LIN {X 0,Y 362.968,Z 415.154,A -85,B 0,C 180,E1 -13446.297,E2 -13446.297} C_VEL
LIN {X 0,Y 357.629,Z 396.824,A -85,B 0,C 180,E1 -13449.531,E2 -13449.531} C_VEL
LIN {X 0,Y 354.805,Z 387.089,A -85,B 0,C 180,E1 -13451.373,E2 -13451.373} C_VEL
LIN {X 0,Y 354.749,Z 386.923,A -85,B 0,C 180,E1 -13454.504,E2 -13454.504} C_VEL
LIN {X 0,Y 354.769,Z 386.876,A -85,B 0,C 180,E1 -13457.659,E2 -13457.659} C_VEL
LIN {X 0,Y 354.773,Z 386.917,A -85,B 0,C 180,E1 -13460.661,E2 -13460.661} C_VEL
LIN {X 0,Y 354.805,Z 386.863,A -85,B 0,C 180,E1 -13464.301,E2 -13464.301} C_VEL
LIN {X 0,Y 354.773,Z 386.912,A -85,B 0,C 180,E1 -13467.665,E2 -13467.665} C_VEL
LIN {X 0,Y 354.785,Z 386.907,A -85,B 0,C 180,E1 -13471.613,E2 -13471.613} C_VEL
LIN {X 0,Y 354.79,Z 386.899,A -85,B 0,C 180,E1 -13475.419,E2 -13475.419} C_VEL
LIN {X 0,Y 354.809,Z 386.903,A -85,B 0,C 180,E1 -13479.112,E2 -13479.112} C_VEL
LIN {X 0,Y 354.836,Z 386.911,A -85,B 0,C 180,E1 -13482.717,E2 -13482.717} C_VEL
LIN {X 0,Y 354.924,Z 386.887,A -85,B 0,C 180,E1 -13486.254,E2 -13486.254} C_VEL
LIN {X 0,Y 354.937,Z 386.882,A -85,B 0,C 180,E1 -13489.735,E2 -13489.735} C_VEL
LIN {X 0,Y 355.066,Z 386.879,A -85,B 0,C 180,E1 -13493.18,E2 -13493.18} C_VEL
LIN {X 0,Y 355.214,Z 386.859,A -85,B 0,C 180,E1 -13497.732,E2 -13497.732} C_VEL
LIN {X 0,Y 355.212,Z 386.849,A -85,B 0,C 180,E1 -13502.268,E2 -13502.268} C_VEL
LIN {X 0,Y 355.089,Z 386.861,A -85,B 0,C 180,E1 -13506.82,E2 -13506.82} C_VEL
LIN {X 0,Y 354.939,Z 386.89,A -85,B 0,C 180,E1 -13510.265,E2 -13510.265} C_VEL
LIN {X 0,Y 354.928,Z 386.895,A -85,B 0,C 180,E1 -13514.019,E2 -13514.019} C_VEL
LIN {X 0,Y 354.876,Z 386.898,A -85,B 0,C 180,E1 -13518.093,E2 -13518.093} C_VEL
LIN {X 0,Y 354.793,Z 386.906,A -85,B 0,C 180,E1 -13522.109,E2 -13522.109} C_VEL
LIN {X 0,Y 354.787,Z 386.904,A -85,B 0,C 180,E1 -13525.836,E2 -13525.836} C_VEL
LIN {X 0,Y 354.78,Z 386.909,A -85,B 0,C 180,E1 -13529.686,E2 -13529.686} C_VEL
LIN {X 0,Y 354.795,Z 386.915,A -85,B 0,C 180,E1 -13533.703,E2 -13533.703} C_VEL
LIN {X 0,Y 354.78,Z 386.888,A -85,B 0,C 180,E1 -13536.462,E2 -13536.462} C_VEL
LIN {X 0,Y 354.757,Z 386.91,A -85,B 0,C 180,E1 -13539.414,E2 -13539.414} C_VEL
LIN {X 0,Y 354.769,Z 386.891,A -85,B 0,C 180,E1 -13542.867,E2 -13542.867} C_VEL
LIN {X 0,Y 354.797,Z 387.142,A -85,B 0,C 180,E1 -13544.912,E2 -13544.912} C_VEL
LIN {X 0,Y 357.139,Z 393.195,A -85,B 0,C 180,E1 -13546.219,E2 -13546.219} C_VEL
LIN {X 0,Y 362.106,Z 406.376,A -85,B 0,C 180,E1 -13548.824,E2 -13548.824} C_VEL
LIN {X 0,Y 366.575,Z 420.211,A -85,B 0,C 180,E1 -13551.376,E2 -13551.376} C_VEL
LIN {X 0,Y 370.495,Z 434.136,A -85,B 0,C 180,E1 -13553.779,E2 -13553.779} C_VEL
LIN {X 0,Y 371.189,Z 437.502,A -85,B 0,C 180,E1 -13554.317,E2 -13554.317} C_VEL
LIN {X 0,Y 369.064,Z 461.57,A -85,B 0,C 180,E1 -13557.353,E2 -13557.353} C_VEL
LIN {X 0,Y 368.412,Z 471.572,A -85,B 0,C 180,E1 -13558.53,E2 -13558.53} C_VEL
LIN {X 0,Y 373.171,Z 501.555,A -85,B 0,C 180,E1 -13559.641,E2 -13559.641} C_VEL
LIN {X 0,Y 374.104,Z 509.019,A -85,B 0,C 180,E1 -13559.887,E2 -13559.887} C_VEL
LIN {X 0,Y 370.581,Z 640.588,A -85,B 0,C 180,E1 -13562.469,E2 -13562.469} C_VEL
LIN {X 0,Y 369.736,Z 655.386,A -85,B 0,C 180,E1 -13562.945,E2 -13562.945} C_VEL
LIN {X 0,Y 368.618,Z 669.241,A -85,B 0,C 180,E1 -13563.582,E2 -13563.582} C_VEL
LIN {X 0,Y 367.111,Z 684.092,A -85,B 0,C 180,E1 -13564.497,E2 -13564.497} C_VEL
LIN {X 0,Y 365.467,Z 697.803,A -85,B 0,C 180,E1 -13565.581,E2 -13565.581} C_VEL
LIN {X 0,Y 363.7,Z 710.491,A -85,B 0,C 180,E1 -13566.816,E2 -13566.816} C_VEL
LIN {X 0,Y 361.771,Z 723.288,A -85,B 0,C 180,E1 -13568.342,E2 -13568.342} C_VEL
LIN {X 0,Y 359.982,Z 734.883,A -85,B 0,C 180,E1 -13570.024,E2 -13570.024} C_VEL
LIN {X 0,Y 358.316,Z 744.651,A -85,B 0,C 180,E1 -13571.712,E2 -13571.712} C_VEL
LIN {X 0,Y 356.802,Z 754.205,A -85,B 0,C 180,E1 -13573.701,E2 -13573.701} C_VEL
LIN {X 0,Y 355.593,Z 762.353,A -85,B 0,C 180,E1 -13575.754,E2 -13575.754} C_VEL
LIN {X 0,Y 354.609,Z 769.585,A -85,B 0,C 180,E1 -13577.991,E2 -13577.991} C_VEL
LIN {X 0,Y 353.878,Z 775.478,A -85,B 0,C 180,E1 -13580.283,E2 -13580.283} C_VEL
LIN {X 0,Y 353.528,Z 778.954,A -85,B 0,C 180,E1 -13582.003,E2 -13582.003} C_VEL
LIN {X 0,Y 353.26,Z 782.496,A -85,B 0,C 180,E1 -13584.293,E2 -13584.293} C_VEL
LIN {X 0,Y 353.184,Z 784.838,A -85,B 0,C 180,E1 -13586.579,E2 -13586.579} C_VEL
LIN {X 0,Y 353.144,Z 786.03,A -85,B 0,C 180,E1 -13588.861,E2 -13588.861} C_VEL
LIN {X 0,Y 353.145,Z 786.044,A -85,B 0,C 180,E1 -13591.142,E2 -13591.142} C_VEL
LIN {X 0,Y 353.186,Z 784.909,A -85,B 0,C 180,E1 -13593.424,E2 -13593.424} C_VEL
LIN {X 0,Y 353.315,Z 782.299,A -85,B 0,C 180,E1 -13595.967,E2 -13595.967} C_VEL
LIN {X 0,Y 353.646,Z 778.076,A -85,B 0,C 180,E1 -13598.573,E2 -13598.573} C_VEL
LIN {X 0,Y 354.128,Z 772.946,A -85,B 0,C 180,E1 -13600.869,E2 -13600.869} C_VEL
LIN {X 0,Y 355.058,Z 766.383,A -85,B 0,C 180,E1 -13603.159,E2 -13603.159} C_VEL
LIN {X 0,Y 355.51,Z 763.086,A -85,B 0,C 180,E1 -13604.138,E2 -13604.138} C_VEL
LIN {X 0,Y 355.295,Z 760.19,A -85,B 0,C 180,E1 -13604.968,E2 -13604.968} C_VEL
LIN {X 0,Y 353.242,Z 755.303,A -85,B 0,C 180,E1 -13606.325,E2 -13606.325} C_VEL
LIN {X 0,Y 351.29,Z 749.969,A -85,B 0,C 180,E1 -13607.649,E2 -13607.649} C_VEL
LIN {X 0,Y 351.23,Z 746.373,A -85,B 0,C 180,E1 -13608.414,E2 -13608.414} C_VEL
LIN {X 0,Y 353.087,Z 735.857,A -85,B 0,C 180,E1 -13610.314,E2 -13610.314} C_VEL
LIN {X 0,Y 355.017,Z 723.948,A -85,B 0,C 180,E1 -13612.096,E2 -13612.096} C_VEL
LIN {X 0,Y 357.067,Z 711.288,A -85,B 0,C 180,E1 -13613.644,E2 -13613.644} C_VEL
LIN {X 0,Y 358.867,Z 698.787,A -85,B 0,C 180,E1 -13614.903,E2 -13614.903} C_VEL
LIN {X 0,Y 360.715,Z 684.652,A -85,B 0,C 180,E1 -13616.046,E2 -13616.046} C_VEL
LIN {X 0,Y 362.175,Z 670.066,A -85,B 0,C 180,E1 -13616.975,E2 -13616.975} C_VEL
LIN {X 0,Y 363.457,Z 655.655,A -85,B 0,C 180,E1 -13617.652,E2 -13617.652} C_VEL
LIN {X 0,Y 364.353,Z 639.939,A -85,B 0,C 180,E1 -13618.164,E2 -13618.164} C_VEL
LIN {X 0,Y 367.302,Z 535.361,A -85,B 0,C 180,E1 -13620.246,E2 -13620.246} C_VEL
LIN {X 0,Y 367.924,Z 508.361,A -85,B 0,C 180,E1 -13620.791,E2 -13620.791} C_VEL
LIN {X 0,Y 362.697,Z 474.811,A -85,B 0,C 180,E1 -13622.047,E2 -13622.047} C_VEL
LIN {X 0,Y 362.119,Z 471.033,A -85,B 0,C 180,E1 -13622.221,E2 -13622.221} C_VEL
LIN {X 0,Y 364.049,Z 448.22,A -85,B 0,C 180,E1 -13625.054,E2 -13625.054} C_VEL
LIN {X 0,Y 364.792,Z 439.692,A -85,B 0,C 180,E1 -13626.166,E2 -13626.166} C_VEL
LIN {X 0,Y 361.536,Z 427.166,A -85,B 0,C 180,E1 -13628.32,E2 -13628.32} C_VEL
LIN {X 0,Y 357.787,Z 414.84,A -85,B 0,C 180,E1 -13630.571,E2 -13630.571} C_VEL
LIN {X 0,Y 352.853,Z 400.954,A -85,B 0,C 180,E1 -13633.326,E2 -13633.326} C_VEL
LIN {X 0,Y 347.745,Z 388.016,A -85,B 0,C 180,E1 -13636.095,E2 -13636.095} C_VEL
LIN {X 0,Y 347.712,Z 387.785,A -85,B 0,C 180,E1 -13638.406,E2 -13638.406} C_VEL
LIN {X 0,Y 347.766,Z 387.788,A -85,B 0,C 180,E1 -13642.015,E2 -13642.015} C_VEL
LIN {X 0,Y 347.748,Z 387.758,A -85,B 0,C 180,E1 -13645.536,E2 -13645.536} C_VEL
LIN {X 0,Y 347.735,Z 387.795,A -85,B 0,C 180,E1 -13648.299,E2 -13648.299} C_VEL
LIN {X 0,Y 347.746,Z 387.792,A -85,B 0,C 180,E1 -13650.985,E2 -13650.985} C_VEL
LIN {X 0,Y 347.793,Z 387.981,A -85,B 0,C 180,E1 -13652.376,E2 -13652.376} C_VEL
LIN {X 0,Y 348.722,Z 391.932,A -85,B 0,C 180,E1 -13653.247,E2 -13653.247} C_VEL
LIN {X 0,Y 359.484,Z 420.146,A -85,B 0,C 180,E1 -13654.74,E2 -13654.74} C_VEL
LIN {X 0,Y 355.715,Z 535.123,A -85,B 0,C 180,E1 -13657.837,E2 -13657.837} C_VEL
LIN {X 0,Y 355.227,Z 550.727,A -85,B 0,C 180,E1 -13658.488,E2 -13658.488} C_VEL
LIN {X 0,Y 354.603,Z 565.332,A -85,B 0,C 180,E1 -13659.327,E2 -13659.327} C_VEL
LIN {X 0,Y 353.691,Z 579.963,A -85,B 0,C 180,E1 -13660.408,E2 -13660.408} C_VEL
LIN {X 0,Y 352.843,Z 593.82,A -85,B 0,C 180,E1 -13661.717,E2 -13661.717} C_VEL
LIN {X 0,Y 351.84,Z 606.827,A -85,B 0,C 180,E1 -13663.223,E2 -13663.223} C_VEL
LIN {X 0,Y 351.135,Z 616.893,A -85,B 0,C 180,E1 -13664.628,E2 -13664.628} C_VEL
LIN {X 0,Y 350.183,Z 627.379,A -85,B 0,C 180,E1 -13666.36,E2 -13666.36} C_VEL
LIN {X 0,Y 349.57,Z 636.146,A -85,B 0,C 180,E1 -13668.108,E2 -13668.108} C_VEL
LIN {X 0,Y 348.967,Z 644.601,A -85,B 0,C 180,E1 -13670.143,E2 -13670.143} C_VEL
LIN {X 0,Y 348.594,Z 650.5,A -85,B 0,C 180,E1 -13671.887,E2 -13671.887} C_VEL
LIN {X 0,Y 348.334,Z 655.341,A -85,B 0,C 180,E1 -13673.629,E2 -13673.629} C_VEL
LIN {X 0,Y 347.977,Z 660.381,A -85,B 0,C 180,E1 -13675.946,E2 -13675.946} C_VEL
LIN {X 0,Y 347.967,Z 663.099,A -85,B 0,C 180,E1 -13677.685,E2 -13677.685} C_VEL
LIN {X 0,Y 348.047,Z 665.484,A -85,B 0,C 180,E1 -13680,E2 -13680} C_VEL
LIN {X 0,Y 348.502,Z 666.421,A -85,B 0,C 180,E1 -13682.311,E2 -13682.311} C_VEL
LIN {X 0,Y 349.06,Z 665.935,A -85,B 0,C 180,E1 -13684.619,E2 -13684.619} C_VEL
LIN {X 0,Y 349.703,Z 664.039,A -85,B 0,C 180,E1 -13686.926,E2 -13686.926} C_VEL
LIN {X 0,Y 350.82,Z 660.596,A -85,B 0,C 180,E1 -13689.222,E2 -13689.222} C_VEL
LIN {X 0,Y 351.834,Z 657.006,A -85,B 0,C 180,E1 -13690.939,E2 -13690.939} C_VEL
LIN {X 0,Y 353.413,Z 650.686,A -85,B 0,C 180,E1 -13693.22,E2 -13693.22} C_VEL
LIN {X 0,Y 354.959,Z 643.625,A -85,B 0,C 180,E1 -13695.209,E2 -13695.209} C_VEL
LIN {X 0,Y 356.859,Z 634.78,A -85,B 0,C 180,E1 -13697.182,E2 -13697.182} C_VEL
LIN {X 0,Y 358.664,Z 625.61,A -85,B 0,C 180,E1 -13698.864,E2 -13698.864} C_VEL
LIN {X 0,Y 360.446,Z 615.653,A -85,B 0,C 180,E1 -13700.368,E2 -13700.368} C_VEL
LIN {X 0,Y 362.343,Z 603.197,A -85,B 0,C 180,E1 -13701.924,E2 -13701.924} C_VEL
LIN {X 0,Y 364.021,Z 591.036,A -85,B 0,C 180,E1 -13703.164,E2 -13703.164} C_VEL
LIN {X 0,Y 365.637,Z 577.686,A -85,B 0,C 180,E1 -13704.258,E2 -13704.258} C_VEL
LIN {X 0,Y 366.991,Z 564.198,A -85,B 0,C 180,E1 -13705.15,E2 -13705.15} C_VEL
LIN {X 0,Y 368.094,Z 548.734,A -85,B 0,C 180,E1 -13705.927,E2 -13705.927} C_VEL
LIN {X 0,Y 369.757,Z 525.884,A -85,B 0,C 180,E1 -13706.796,E2 -13706.796} C_VEL
LIN {X 0,Y 377.897,Z 451.52,A -85,B 0,C 180,E1 -13709.427,E2 -13709.427} C_VEL
LIN {X 0,Y 378.713,Z 443.174,A -85,B 0,C 180,E1 -13709.753,E2 -13709.753} C_VEL
LIN {X 0,Y 374.725,Z 436.391,A -85,B 0,C 180,E1 -13711.04,E2 -13711.04} C_VEL
LIN {X 0,Y 370.277,Z 430.062,A -85,B 0,C 180,E1 -13712.635,E2 -13712.635} C_VEL
LIN {X 0,Y 366.994,Z 426.007,A -85,B 0,C 180,E1 -13713.98,E2 -13713.98} C_VEL
LIN {X 0,Y 364.266,Z 422.895,A -85,B 0,C 180,E1 -13715.295,E2 -13715.295} C_VEL
LIN {X 0,Y 361.379,Z 419.769,A -85,B 0,C 180,E1 -13717.12,E2 -13717.12} C_VEL
LIN {X 0,Y 361.362,Z 419.182,A -85,B 0,C 180,E1 -13718.925,E2 -13718.925} C_VEL
LIN {X 0,Y 361.655,Z 419.554,A -85,B 0,C 180,E1 -13721.355,E2 -13721.355} C_VEL
LIN {X 0,Y 362.637,Z 421.568,A -85,B 0,C 180,E1 -13724.242,E2 -13724.242} C_VEL
LIN {X 0,Y 363.768,Z 424.413,A -85,B 0,C 180,E1 -13726.426,E2 -13726.426} C_VEL
LIN {X 0,Y 365.158,Z 428.525,A -85,B 0,C 180,E1 -13728.643,E2 -13728.643} C_VEL
LIN {X 0,Y 366.624,Z 433.697,A -85,B 0,C 180,E1 -13730.757,E2 -13730.757} C_VEL
LIN {X 0,Y 368.039,Z 439.973,A -85,B 0,C 180,E1 -13732.763,E2 -13732.763} C_VEL
LIN {X 0,Y 370.061,Z 445.463,A -85,B 0,C 180,E1 -13733.732,E2 -13733.732} C_VEL
LIN {X 0,Y 371.308,Z 455.894,A -85,B 0,C 180,E1 -13734.7,E2 -13734.7} C_VEL
LIN {X 0,Y 372.834,Z 472.254,A -85,B 0,C 180,E1 -13735.965,E2 -13735.965} C_VEL
LIN {X 0,Y 373.775,Z 487.634,A -85,B 0,C 180,E1 -13736.955,E2 -13736.955} C_VEL
LIN {X 0,Y 374.116,Z 504.327,A -85,B 0,C 180,E1 -13737.835,E2 -13737.835} C_VEL
LIN {X 0,Y 373.957,Z 509.719,A -85,B 0,C 180,E1 -13738.061,E2 -13738.061} C_VEL
LIN {X 0,Y 368.616,Z 574.67,A -85,B 0,C 180,E1 -13740.085,E2 -13740.085} C_VEL
LIN {X 0,Y 365.731,Z 612.624,A -85,B 0,C 180,E1 -13741.247,E2 -13741.247} C_VEL
LIN {X 0,Y 364.27,Z 626.12,A -85,B 0,C 180,E1 -13741.79,E2 -13741.79} C_VEL
LIN {X 0,Y 363.515,Z 645.43,A -85,B 0,C 180,E1 -13742.235,E2 -13742.235} C_VEL
LIN {X 0,Y 362.466,Z 660.753,A -85,B 0,C 180,E1 -13742.814,E2 -13742.814} C_VEL
LIN {X 0,Y 361.182,Z 674.979,A -85,B 0,C 180,E1 -13743.57,E2 -13743.57} C_VEL
LIN {X 0,Y 359.668,Z 688.894,A -85,B 0,C 180,E1 -13744.538,E2 -13744.538} C_VEL
LIN {X 0,Y 357.77,Z 703.113,A -85,B 0,C 180,E1 -13745.789,E2 -13745.789} C_VEL
LIN {X 0,Y 355.877,Z 715.961,A -85,B 0,C 180,E1 -13747.196,E2 -13747.196} C_VEL
LIN {X 0,Y 353.992,Z 727.703,A -85,B 0,C 180,E1 -13748.755,E2 -13748.755} C_VEL
LIN {X 0,Y 352.295,Z 738.439,A -85,B 0,C 180,E1 -13750.478,E2 -13750.478} C_VEL
LIN {X 0,Y 350.726,Z 747.527,A -85,B 0,C 180,E1 -13752.205,E2 -13752.205} C_VEL
LIN {X 0,Y 349.286,Z 756.423,A -85,B 0,C 180,E1 -13754.237,E2 -13754.237} C_VEL
LIN {X 0,Y 348.026,Z 764.73,A -85,B 0,C 180,E1 -13756.57,E2 -13756.57} C_VEL
LIN {X 0,Y 347.132,Z 771.379,A -85,B 0,C 180,E1 -13758.909,E2 -13758.909} C_VEL
LIN {X 0,Y 346.628,Z 776.575,A -85,B 0,C 180,E1 -13761.252,E2 -13761.252} C_VEL
LIN {X 0,Y 346.325,Z 780.853,A -85,B 0,C 180,E1 -13763.912,E2 -13763.912} C_VEL
LIN {X 0,Y 346.187,Z 783.505,A -85,B 0,C 180,E1 -13766.507,E2 -13766.507} C_VEL
LIN {X 0,Y 346.129,Z 784.673,A -85,B 0,C 180,E1 -13768.835,E2 -13768.835} C_VEL
LIN {X 0,Y 346.132,Z 784.671,A -85,B 0,C 180,E1 -13771.162,E2 -13771.162} C_VEL
LIN {X 0,Y 346.189,Z 783.496,A -85,B 0,C 180,E1 -13773.49,E2 -13773.49} C_VEL
LIN {X 0,Y 346.285,Z 780.913,A -85,B 0,C 180,E1 -13776.026,E2 -13776.026} C_VEL
LIN {X 0,Y 346.621,Z 776.563,A -85,B 0,C 180,E1 -13778.745,E2 -13778.745} C_VEL
LIN {X 0,Y 347.125,Z 771.36,A -85,B 0,C 180,E1 -13781.087,E2 -13781.087} C_VEL
LIN {X 0,Y 348.009,Z 764.698,A -85,B 0,C 180,E1 -13783.427,E2 -13783.427} C_VEL
LIN {X 0,Y 349.267,Z 756.386,A -85,B 0,C 180,E1 -13785.76,E2 -13785.76} C_VEL
LIN {X 0,Y 350.692,Z 747.486,A -85,B 0,C 180,E1 -13787.793,E2 -13787.793} C_VEL
LIN {X 0,Y 352.266,Z 738.387,A -85,B 0,C 180,E1 -13789.52,E2 -13789.52} C_VEL
LIN {X 0,Y 353.967,Z 727.642,A -85,B 0,C 180,E1 -13791.243,E2 -13791.243} C_VEL
LIN {X 0,Y 355.824,Z 715.892,A -85,B 0,C 180,E1 -13792.804,E2 -13792.804} C_VEL
LIN {X 0,Y 357.747,Z 703.017,A -85,B 0,C 180,E1 -13794.208,E2 -13794.208} C_VEL
LIN {X 0,Y 359.399,Z 690.514,A -85,B 0,C 180,E1 -13795.323,E2 -13795.323} C_VEL
LIN {X 0,Y 361.03,Z 676.025,A -85,B 0,C 180,E1 -13796.355,E2 -13796.355} C_VEL
LIN {X 0,Y 362.375,Z 661.307,A -85,B 0,C 180,E1 -13797.151,E2 -13797.151} C_VEL
LIN {X 0,Y 363.412,Z 646.234,A -85,B 0,C 180,E1 -13797.73,E2 -13797.73} C_VEL
LIN {X 0,Y 364.103,Z 629.144,A -85,B 0,C 180,E1 -13798.142,E2 -13798.142} C_VEL
LIN {X 0,Y 367.019,Z 518.003,A -85,B 0,C 180,E1 -13800.331,E2 -13800.331} C_VEL
LIN {X 0,Y 367.175,Z 504.545,A -85,B 0,C 180,E1 -13800.615,E2 -13800.615} C_VEL
LIN {X 0,Y 363.359,Z 473.493,A -85,B 0,C 180,E1 -13801.676,E2 -13801.676} C_VEL
LIN {X 0,Y 362.286,Z 465.651,A -85,B 0,C 180,E1 -13801.993,E2 -13801.993} C_VEL
LIN {X 0,Y 360.716,Z 438.296,A -85,B 0,C 180,E1 -13803.739,E2 -13803.739} C_VEL
LIN {X 0,Y 359.932,Z 430.462,A -85,B 0,C 180,E1 -13804.261,E2 -13804.261} C_VEL
LIN {X 0,Y 355.292,Z 413.79,A -85,B 0,C 180,E1 -13807.067,E2 -13807.067} C_VEL
LIN {X 0,Y 350.111,Z 396.023,A -85,B 0,C 180,E1 -13810.289,E2 -13810.289} C_VEL
LIN {X 0,Y 347.758,Z 387.949,A -85,B 0,C 180,E1 -13811.875,E2 -13811.875} C_VEL
LIN {X 0,Y 347.691,Z 387.801,A -85,B 0,C 180,E1 -13815.026,E2 -13815.026} C_VEL
LIN {X 0,Y 347.725,Z 387.754,A -85,B 0,C 180,E1 -13818.398,E2 -13818.398} C_VEL
LIN {X 0,Y 347.749,Z 387.784,A -85,B 0,C 180,E1 -13822.013,E2 -13822.013} C_VEL
LIN {X 0,Y 347.729,Z 387.746,A -85,B 0,C 180,E1 -13825.535,E2 -13825.535} C_VEL
LIN {X 0,Y 347.732,Z 387.794,A -85,B 0,C 180,E1 -13828.299,E2 -13828.299} C_VEL
LIN {X 0,Y 347.731,Z 387.781,A -85,B 0,C 180,E1 -13830.983,E2 -13830.983} C_VEL
LIN {X 0,Y 347.729,Z 387.794,A -85,B 0,C 180,E1 -13833.599,E2 -13833.599} C_VEL
LIN {X 0,Y 347.734,Z 387.782,A -85,B 0,C 180,E1 -13836.158,E2 -13836.158} C_VEL
LIN {X 0,Y 347.761,Z 387.774,A -85,B 0,C 180,E1 -13839.906,E2 -13839.906} C_VEL
LIN {X 0,Y 347.782,Z 387.786,A -85,B 0,C 180,E1 -13843.566,E2 -13843.566} C_VEL
LIN {X 0,Y 347.871,Z 387.777,A -85,B 0,C 180,E1 -13847.16,E2 -13847.16} C_VEL
LIN {X 0,Y 347.919,Z 387.753,A -85,B 0,C 180,E1 -13850.7,E2 -13850.7} C_VEL
LIN {X 0,Y 348.019,Z 387.752,A -85,B 0,C 180,E1 -13854.205,E2 -13854.205} C_VEL
LIN {X 0,Y 348.176,Z 387.735,A -85,B 0,C 180,E1 -13857.686,E2 -13857.686} C_VEL
LIN {X 0,Y 348.127,Z 387.725,A -85,B 0,C 180,E1 -13861.157,E2 -13861.157} C_VEL
LIN {X 0,Y 348.174,Z 387.726,A -85,B 0,C 180,E1 -13862.314,E2 -13862.314} C_VEL
LIN {X 0,Y 348.057,Z 387.736,A -85,B 0,C 180,E1 -13866.959,E2 -13866.959} C_VEL
LIN {X 0,Y 347.879,Z 387.765,A -85,B 0,C 180,E1 -13870.476,E2 -13870.476} C_VEL
LIN {X 0,Y 347.884,Z 387.773,A -85,B 0,C 180,E1 -13874.151,E2 -13874.151} C_VEL
LIN {X 0,Y 347.815,Z 387.779,A -85,B 0,C 180,E1 -13878.26,E2 -13878.26} C_VEL
LIN {X 0,Y 347.75,Z 387.778,A -85,B 0,C 180,E1 -13881.625,E2 -13881.625} C_VEL
LIN {X 0,Y 347.724,Z 387.783,A -85,B 0,C 180,E1 -13885.115,E2 -13885.115} C_VEL
LIN {X 0,Y 347.711,Z 387.798,A -85,B 0,C 180,E1 -13887.703,E2 -13887.703} C_VEL
LIN {X 0,Y 347.716,Z 387.794,A -85,B 0,C 180,E1 -13890.351,E2 -13890.351} C_VEL
LIN {X 0,Y 347.736,Z 387.797,A -85,B 0,C 180,E1 -13894.045,E2 -13894.045} C_VEL
LIN {X 0,Y 347.742,Z 387.757,A -85,B 0,C 180,E1 -13897.323,E2 -13897.323} C_VEL
LIN {X 0,Y 347.685,Z 387.803,A -85,B 0,C 180,E1 -13900.304,E2 -13900.304} C_VEL
LIN {X 0,Y 347.706,Z 387.802,A -85,B 0,C 180,E1 -13903.811,E2 -13903.811} C_VEL
LIN {X 0,Y 347.837,Z 388.477,A -85,B 0,C 180,E1 -13904.167,E2 -13904.167} C_VEL
LIN {X 0,Y 353.36,Z 402.251,A -85,B 0,C 180,E1 -13907.078,E2 -13907.078} C_VEL
LIN {X 0,Y 357.842,Z 415.141,A -85,B 0,C 180,E1 -13909.603,E2 -13909.603} C_VEL
LIN {X 0,Y 362.251,Z 429.616,A -85,B 0,C 180,E1 -13912.24,E2 -13912.24} C_VEL
LIN {X 0,Y 364.709,Z 439.031,A -85,B 0,C 180,E1 -13913.847,E2 -13913.847} C_VEL
LIN {X 0,Y 362.977,Z 460.412,A -85,B 0,C 180,E1 -13916.599,E2 -13916.599} C_VEL
LIN {X 0,Y 362.114,Z 471.362,A -85,B 0,C 180,E1 -13917.912,E2 -13917.912} C_VEL
LIN {X 0,Y 367.095,Z 502.828,A -85,B 0,C 180,E1 -13919.115,E2 -13919.115} C_VEL
LIN {X 0,Y 367.958,Z 510.239,A -85,B 0,C 180,E1 -13919.36,E2 -13919.36} C_VEL
LIN {X 0,Y 364.305,Z 640.508,A -85,B 0,C 180,E1 -13921.953,E2 -13921.953} C_VEL
LIN {X 0,Y 363.444,Z 655.334,A -85,B 0,C 180,E1 -13922.437,E2 -13922.437} C_VEL
LIN {X 0,Y 362.258,Z 669.202,A -85,B 0,C 180,E1 -13923.082,E2 -13923.082} C_VEL
LIN {X 0,Y 360.849,Z 682.671,A -85,B 0,C 180,E1 -13923.91,E2 -13923.91} C_VEL
LIN {X 0,Y 359.206,Z 696.235,A -85,B 0,C 180,E1 -13924.972,E2 -13924.972} C_VEL
LIN {X 0,Y 357.307,Z 709.205,A -85,B 0,C 180,E1 -13926.223,E2 -13926.223} C_VEL
LIN {X 0,Y 355.314,Z 722.219,A -85,B 0,C 180,E1 -13927.775,E2 -13927.775} C_VEL
LIN {X 0,Y 353.583,Z 733.162,A -85,B 0,C 180,E1 -13929.352,E2 -13929.352} C_VEL
LIN {X 0,Y 351.807,Z 743.153,A -85,B 0,C 180,E1 -13931.059,E2 -13931.059} C_VEL
LIN {X 0,Y 350.173,Z 752.964,A -85,B 0,C 180,E1 -13933.083,E2 -13933.083} C_VEL
LIN {X 0,Y 348.7,Z 761.909,A -85,B 0,C 180,E1 -13935.338,E2 -13935.338} C_VEL
LIN {X 0,Y 347.635,Z 769.57,A -85,B 0,C 180,E1 -13937.746,E2 -13937.746} C_VEL
LIN {X 0,Y 346.835,Z 775.464,A -85,B 0,C 180,E1 -13940.084,E2 -13940.084} C_VEL
LIN {X 0,Y 346.481,Z 778.94,A -85,B 0,C 180,E1 -13941.839,E2 -13941.839} C_VEL
LIN {X 0,Y 346.18,Z 782.483,A -85,B 0,C 180,E1 -13944.176,E2 -13944.176} C_VEL
LIN {X 0,Y 346.109,Z 784.824,A -85,B 0,C 180,E1 -13946.509,E2 -13946.509} C_VEL
LIN {X 0,Y 346.047,Z 786.016,A -85,B 0,C 180,E1 -13948.838,E2 -13948.838} C_VEL
LIN {X 0,Y 346.048,Z 786.03,A -85,B 0,C 180,E1 -13951.166,E2 -13951.166} C_VEL
LIN {X 0,Y 346.111,Z 784.895,A -85,B 0,C 180,E1 -13953.494,E2 -13953.494} C_VEL
LIN {X 0,Y 346.235,Z 782.462,A -85,B 0,C 180,E1 -13955.945,E2 -13955.945} C_VEL
LIN {X 0,Y 346.497,Z 779.115,A -85,B 0,C 180,E1 -13958.164,E2 -13958.164} C_VEL
LIN {X 0,Y 346.949,Z 774.338,A -85,B 0,C 180,E1 -13960.506,E2 -13960.506} C_VEL
LIN {X 0,Y 347.855,Z 768.153,A -85,B 0,C 180,E1 -13962.842,E2 -13962.842} C_VEL
LIN {X 0,Y 348.928,Z 760.373,A -85,B 0,C 180,E1 -13965.181,E2 -13965.181} C_VEL
LIN {X 0,Y 350.3,Z 752.075,A -85,B 0,C 180,E1 -13967.215,E2 -13967.215} C_VEL
LIN {X 0,Y 351.23,Z 746.373,A -85,B 0,C 180,E1 -13968.414,E2 -13968.414} C_VEL
LIN {X 0,Y 351.226,Z 742.681,A -85,B 0,C 180,E1 -13969.166,E2 -13969.166} C_VEL
LIN {X 0,Y 349.58,Z 736.566,A -85,B 0,C 180,E1 -13970.42,E2 -13970.42} C_VEL
LIN {X 0,Y 348.006,Z 730.079,A -85,B 0,C 180,E1 -13971.624,E2 -13971.624} C_VEL
LIN {X 0,Y 348.097,Z 725.756,A -85,B 0,C 180,E1 -13972.286,E2 -13972.286} C_VEL
LIN {X 0,Y 350.184,Z 713.786,A -85,B 0,C 180,E1 -13973.824,E2 -13973.824} C_VEL
LIN {X 0,Y 351.975,Z 701.811,A -85,B 0,C 180,E1 -13975.108,E2 -13975.108} C_VEL
LIN {X 0,Y 353.936,Z 688.178,A -85,B 0,C 180,E1 -13976.286,E2 -13976.286} C_VEL
LIN {X 0,Y 355.528,Z 673.717,A -85,B 0,C 180,E1 -13977.283,E2 -13977.283} C_VEL
LIN {X 0,Y 356.899,Z 658.985,A -85,B 0,C 180,E1 -13978.045,E2 -13978.045} C_VEL
LIN {X 0,Y 357.946,Z 643.838,A -85,B 0,C 180,E1 -13978.595,E2 -13978.595} C_VEL
LIN {X 0,Y 358.77,Z 619.75,A -85,B 0,C 180,E1 -13979.123,E2 -13979.123} C_VEL
LIN {X 0,Y 361.905,Z 509.972,A -85,B 0,C 180,E1 -13981.32,E2 -13981.32} C_VEL
LIN {X 0,Y 356.745,Z 476.476,A -85,B 0,C 180,E1 -13982.604,E2 -13982.604} C_VEL
LIN {X 0,Y 355.921,Z 471.37,A -85,B 0,C 180,E1 -13982.82,E2 -13982.82} C_VEL
LIN {X 0,Y 357.59,Z 451.723,A -85,B 0,C 180,E1 -13985.265,E2 -13985.265} C_VEL
LIN {X 0,Y 358.467,Z 442.195,A -85,B 0,C 180,E1 -13986.502,E2 -13986.502} C_VEL
LIN {X 0,Y 354.759,Z 428.17,A -85,B 0,C 180,E1 -13988.962,E2 -13988.962} C_VEL
LIN {X 0,Y 351.384,Z 417.222,A -85,B 0,C 180,E1 -13991.021,E2 -13991.021} C_VEL
LIN {X 0,Y 347.08,Z 404.93,A -85,B 0,C 180,E1 -13993.51,E2 -13993.51} C_VEL
LIN {X 0,Y 341.543,Z 391.259,A -85,B 0,C 180,E1 -13996.456,E2 -13996.456} C_VEL
LIN {X 0,Y 340.688,Z 388.832,A -85,B 0,C 180,E1 -13997.073,E2 -13997.073} C_VEL
LIN {X 0,Y 340.66,Z 388.647,A -85,B 0,C 180,E1 -14000.242,E2 -14000.242} C_VEL
LIN {X 0,Y 340.711,Z 388.652,A -85,B 0,C 180,E1 -14003.561,E2 -14003.561} C_VEL
LIN {X 0,Y 340.695,Z 388.641,A -85,B 0,C 180,E1 -14006.154,E2 -14006.154} C_VEL
LIN {X 0,Y 340.722,Z 388.67,A -85,B 0,C 180,E1 -14010.037,E2 -14010.037} C_VEL
LIN {X 0,Y 340.716,Z 388.834,A -85,B 0,C 180,E1 -14011.985,E2 -14011.985} C_VEL
LIN {X 0,Y 341.513,Z 392.232,A -85,B 0,C 180,E1 -14012.791,E2 -14012.791} C_VEL
LIN {X 0,Y 352.608,Z 421.381,A -85,B 0,C 180,E1 -14014.388,E2 -14014.388} C_VEL
LIN {X 0,Y 352.505,Z 430.153,A -85,B 0,C 180,E1 -14014.641,E2 -14014.641} C_VEL
LIN {X 0,Y 348.862,Z 535.67,A -85,B 0,C 180,E1 -14017.553,E2 -14017.553} C_VEL
LIN {X 0,Y 348.355,Z 551.577,A -85,B 0,C 180,E1 -14018.231,E2 -14018.231} C_VEL
LIN {X 0,Y 347.656,Z 566.805,A -85,B 0,C 180,E1 -14019.127,E2 -14019.127} C_VEL
LIN {X 0,Y 346.776,Z 580.423,A -85,B 0,C 180,E1 -14020.155,E2 -14020.155} C_VEL
LIN {X 0,Y 346.029,Z 593.034,A -85,B 0,C 180,E1 -14021.344,E2 -14021.344} C_VEL
LIN {X 0,Y 345.006,Z 605.891,A -85,B 0,C 180,E1 -14022.82,E2 -14022.82} C_VEL
LIN {X 0,Y 344.229,Z 616.863,A -85,B 0,C 180,E1 -14024.342,E2 -14024.342} C_VEL
LIN {X 0,Y 343.224,Z 627.349,A -85,B 0,C 180,E1 -14026.078,E2 -14026.078} C_VEL
LIN {X 0,Y 342.608,Z 636.286,A -85,B 0,C 180,E1 -14027.862,E2 -14027.862} C_VEL
LIN {X 0,Y 341.976,Z 644.907,A -85,B 0,C 180,E1 -14029.94,E2 -14029.94} C_VEL
LIN {X 0,Y 341.557,Z 650.942,A -85,B 0,C 180,E1 -14031.719,E2 -14031.719} C_VEL
LIN {X 0,Y 341.306,Z 655.934,A -85,B 0,C 180,E1 -14033.497,E2 -14033.497} C_VEL
LIN {X 0,Y 340.865,Z 660.025,A -85,B 0,C 180,E1 -14035.269,E2 -14035.269} C_VEL
LIN {X 0,Y 341.006,Z 662.178,A -85,B 0,C 180,E1 -14036.455,E2 -14036.455} C_VEL
LIN {X 0,Y 341.003,Z 665.418,A -85,B 0,C 180,E1 -14038.819,E2 -14038.819} C_VEL
LIN {X 0,Y 341.257,Z 667.212,A -85,B 0,C 180,E1 -14041.18,E2 -14041.18} C_VEL
LIN {X 0,Y 341.82,Z 667.567,A -85,B 0,C 180,E1 -14043.536,E2 -14043.536} C_VEL
LIN {X 0,Y 342.413,Z 666.541,A -85,B 0,C 180,E1 -14045.89,E2 -14045.89} C_VEL
LIN {X 0,Y 343.413,Z 664.023,A -85,B 0,C 180,E1 -14048.236,E2 -14048.236} C_VEL
LIN {X 0,Y 344.633,Z 659.991,A -85,B 0,C 180,E1 -14050.576,E2 -14050.576} C_VEL
LIN {X 0,Y 345.862,Z 655.892,A -85,B 0,C 180,E1 -14052.328,E2 -14052.328} C_VEL
LIN {X 0,Y 347.199,Z 650.782,A -85,B 0,C 180,E1 -14054.058,E2 -14054.058} C_VEL
LIN {X 0,Y 348.972,Z 643.472,A -85,B 0,C 180,E1 -14056.076,E2 -14056.076} C_VEL
LIN {X 0,Y 351.017,Z 634.348,A -85,B 0,C 180,E1 -14058.079,E2 -14058.079} C_VEL
LIN {X 0,Y 353.272,Z 623.585,A -85,B 0,C 180,E1 -14059.967,E2 -14059.967} C_VEL
LIN {X 0,Y 355.251,Z 612.858,A -85,B 0,C 180,E1 -14061.529,E2 -14061.529} C_VEL
LIN {X 0,Y 357.071,Z 601.633,A -85,B 0,C 180,E1 -14062.875,E2 -14062.875} C_VEL
LIN {X 0,Y 358.899,Z 588.957,A -85,B 0,C 180,E1 -14064.128,E2 -14064.128} C_VEL
LIN {X 0,Y 360.624,Z 574.998,A -85,B 0,C 180,E1 -14065.233,E2 -14065.233} C_VEL
LIN {X 0,Y 362.049,Z 560.556,A -85,B 0,C 180,E1 -14066.13,E2 -14066.13} C_VEL
LIN {X 0,Y 363.173,Z 544.943,A -85,B 0,C 180,E1 -14066.874,E2 -14066.874} C_VEL
LIN {X 0,Y 367.035,Z 505.116,A -85,B 0,C 180,E1 -14068.366,E2 -14068.366} C_VEL
LIN {X 0,Y 374.148,Z 446.937,A -85,B 0,C 180,E1 -14070.475,E2 -14070.475} C_VEL
LIN {X 0,Y 370.251,Z 440.38,A -85,B 0,C 180,E1 -14071.854,E2 -14071.854} C_VEL
LIN {X 0,Y 366.701,Z 435.364,A -85,B 0,C 180,E1 -14073.249,E2 -14073.249} C_VEL
LIN {X 0,Y 364.316,Z 432.271,A -85,B 0,C 180,E1 -14074.315,E2 -14074.315} C_VEL
LIN {X 0,Y 361.669,Z 429.229,A -85,B 0,C 180,E1 -14075.659,E2 -14075.659} C_VEL
LIN {X 0,Y 358.847,Z 426.243,A -85,B 0,C 180,E1 -14077.481,E2 -14077.481} C_VEL
LIN {X 0,Y 356.486,Z 424.249,A -85,B 0,C 180,E1 -14079.746,E2 -14079.746} C_VEL
LIN {X 0,Y 356.251,Z 424.05,A -85,B 0,C 180,E1 -14080.618,E2 -14080.618} C_VEL
LIN {X 0,Y 356.92,Z 425.459,A -85,B 0,C 180,E1 -14083.233,E2 -14083.233} C_VEL
LIN {X 0,Y 357.699,Z 427.225,A -85,B 0,C 180,E1 -14085.017,E2 -14085.017} C_VEL
LIN {X 0,Y 358.917,Z 430.509,A -85,B 0,C 180,E1 -14087.246,E2 -14087.246} C_VEL
LIN {X 0,Y 360.339,Z 435.217,A -85,B 0,C 180,E1 -14089.521,E2 -14089.521} C_VEL
LIN {X 0,Y 361.053,Z 437.334,A -85,B 0,C 180,E1 -14090.252,E2 -14090.252} C_VEL
LIN {X 0,Y 364.955,Z 445.882,A -85,B 0,C 180,E1 -14092.365,E2 -14092.365} C_VEL
LIN {X 0,Y 366.418,Z 450.057,A -85,B 0,C 180,E1 -14093.102,E2 -14093.102} C_VEL
LIN {X 0,Y 367.621,Z 463.677,A -85,B 0,C 180,E1 -14094.33,E2 -14094.33} C_VEL
LIN {X 0,Y 368.658,Z 478.531,A -85,B 0,C 180,E1 -14095.465,E2 -14095.465} C_VEL
LIN {X 0,Y 369.269,Z 494.828,A -85,B 0,C 180,E1 -14096.499,E2 -14096.499} C_VEL
LIN {X 0,Y 369.14,Z 509.744,A -85,B 0,C 180,E1 -14097.249,E2 -14097.249} C_VEL
LIN {X 0,Y 363.288,Z 575.199,A -85,B 0,C 180,E1 -14099.359,E2 -14099.359} C_VEL
LIN {X 0,Y 360.231,Z 611.939,A -85,B 0,C 180,E1 -14100.526,E2 -14100.526} C_VEL
LIN {X 0,Y 358.103,Z 628.907,A -85,B 0,C 180,E1 -14101.259,E2 -14101.259} C_VEL
LIN {X 0,Y 357.778,Z 634.992,A -85,B 0,C 180,E1 -14101.431,E2 -14101.431} C_VEL
LIN {X 0,Y 356.918,Z 650.781,A -85,B 0,C 180,E1 -14101.877,E2 -14101.877} C_VEL
LIN {X 0,Y 355.807,Z 665.201,A -85,B 0,C 180,E1 -14102.501,E2 -14102.501} C_VEL
LIN {X 0,Y 354.49,Z 678.829,A -85,B 0,C 180,E1 -14103.302,E2 -14103.302} C_VEL
LIN {X 0,Y 352.844,Z 692.433,A -85,B 0,C 180,E1 -14104.326,E2 -14104.326} C_VEL
LIN {X 0,Y 350.903,Z 705.973,A -85,B 0,C 180,E1 -14105.6,E2 -14105.6} C_VEL
LIN {X 0,Y 348.74,Z 719.461,A -85,B 0,C 180,E1 -14107.172,E2 -14107.172} C_VEL
LIN {X 0,Y 346.855,Z 730.596,A -85,B 0,C 180,E1 -14108.757,E2 -14108.757} C_VEL
LIN {X 0,Y 344.945,Z 741.694,A -85,B 0,C 180,E1 -14110.664,E2 -14110.664} C_VEL
LIN {X 0,Y 343.242,Z 751.579,A -85,B 0,C 180,E1 -14112.727,E2 -14112.727} C_VEL
LIN {X 0,Y 341.709,Z 760.566,A -85,B 0,C 180,E1 -14115.025,E2 -14115.025} C_VEL
LIN {X 0,Y 340.619,Z 768.264,A -85,B 0,C 180,E1 -14117.486,E2 -14117.486} C_VEL
LIN {X 0,Y 339.813,Z 774.164,A -85,B 0,C 180,E1 -14119.873,E2 -14119.873} C_VEL
LIN {X 0,Y 339.486,Z 777.651,A -85,B 0,C 180,E1 -14121.666,E2 -14121.666} C_VEL
LIN {X 0,Y 339.209,Z 781.193,A -85,B 0,C 180,E1 -14124.052,E2 -14124.052} C_VEL
LIN {X 0,Y 339.111,Z 783.52,A -85,B 0,C 180,E1 -14126.434,E2 -14126.434} C_VEL
LIN {X 0,Y 339.032,Z 784.687,A -85,B 0,C 180,E1 -14128.81,E2 -14128.81} C_VEL
LIN {X 0,Y 339.035,Z 784.685,A -85,B 0,C 180,E1 -14131.186,E2 -14131.186} C_VEL
LIN {X 0,Y 339.112,Z 783.51,A -85,B 0,C 180,E1 -14133.563,E2 -14133.563} C_VEL
LIN {X 0,Y 339.204,Z 781.105,A -85,B 0,C 180,E1 -14136.005,E2 -14136.005} C_VEL
LIN {X 0,Y 339.482,Z 777.637,A -85,B 0,C 180,E1 -14138.33,E2 -14138.33} C_VEL
LIN {X 0,Y 339.939,Z 772.793,A -85,B 0,C 180,E1 -14140.721,E2 -14140.721} C_VEL
LIN {X 0,Y 340.845,Z 766.514,A -85,B 0,C 180,E1 -14143.107,E2 -14143.107} C_VEL
LIN {X 0,Y 341.994,Z 758.622,A -85,B 0,C 180,E1 -14145.493,E2 -14145.493} C_VEL
LIN {X 0,Y 343.404,Z 750.195,A -85,B 0,C 180,E1 -14147.568,E2 -14147.568} C_VEL
LIN {X 0,Y 345.233,Z 740.024,A -85,B 0,C 180,E1 -14149.625,E2 -14149.625} C_VEL
LIN {X 0,Y 346.98,Z 729.601,A -85,B 0,C 180,E1 -14151.38,E2 -14151.38} C_VEL
LIN {X 0,Y 348.885,Z 718.245,A -85,B 0,C 180,E1 -14152.97,E2 -14152.97} C_VEL
LIN {X 0,Y 350.845,Z 705.874,A -85,B 0,C 180,E1 -14154.401,E2 -14154.401} C_VEL
LIN {X 0,Y 352.765,Z 692.293,A -85,B 0,C 180,E1 -14155.676,E2 -14155.676} C_VEL
LIN {X 0,Y 354.501,Z 677.732,A -85,B 0,C 180,E1 -14156.76,E2 -14156.76} C_VEL
LIN {X 0,Y 355.952,Z 662.855,A -85,B 0,C 180,E1 -14157.603,E2 -14157.603} C_VEL
LIN {X 0,Y 357.042,Z 648.533,A -85,B 0,C 180,E1 -14158.189,E2 -14158.189} C_VEL
LIN {X 0,Y 357.772,Z 632.81,A -85,B 0,C 180,E1 -14158.606,E2 -14158.606} C_VEL
LIN {X 0,Y 360.883,Z 520.509,A -85,B 0,C 180,E1 -14160.848,E2 -14160.848} C_VEL
LIN {X 0,Y 361.079,Z 505.255,A -85,B 0,C 180,E1 -14161.176,E2 -14161.176} C_VEL
LIN {X 0,Y 357.05,Z 472.691,A -85,B 0,C 180,E1 -14162.324,E2 -14162.324} C_VEL
LIN {X 0,Y 356.156,Z 465.789,A -85,B 0,C 180,E1 -14162.611,E2 -14162.611} C_VEL
LIN {X 0,Y 354.627,Z 436.894,A -85,B 0,C 180,E1 -14164.507,E2 -14164.507} C_VEL
LIN {X 0,Y 354.128,Z 433.29,A -85,B 0,C 180,E1 -14164.77,E2 -14164.77} C_VEL
LIN {X 0,Y 351.09,Z 424.871,A -85,B 0,C 180,E1 -14165.673,E2 -14165.673} C_VEL
LIN {X 0,Y 346.016,Z 407.006,A -85,B 0,C 180,E1 -14168.856,E2 -14168.856} C_VEL
LIN {X 0,Y 340.746,Z 388.881,A -85,B 0,C 180,E1 -14172.338,E2 -14172.338} C_VEL
LIN {X 0,Y 340.638,Z 388.65,A -85,B 0,C 180,E1 -14176.226,E2 -14176.226} C_VEL
LIN {X 0,Y 340.655,Z 388.636,A -85,B 0,C 180,E1 -14178.686,E2 -14178.686} C_VEL
LIN {X 0,Y 340.706,Z 388.665,A -85,B 0,C 180,E1 -14181.769,E2 -14181.769} C_VEL
LIN {X 0,Y 340.709,Z 388.619,A -85,B 0,C 180,E1 -14185.595,E2 -14185.595} C_VEL
LIN {X 0,Y 340.68,Z 388.673,A -85,B 0,C 180,E1 -14188.954,E2 -14188.954} C_VEL
LIN {X 0,Y 340.703,Z 388.671,A -85,B 0,C 180,E1 -14193.011,E2 -14193.011} C_VEL
LIN {X 0,Y 340.686,Z 388.67,A -85,B 0,C 180,E1 -14196.924,E2 -14196.924} C_VEL
LIN {X 0,Y 340.692,Z 388.657,A -85,B 0,C 180,E1 -14200.728,E2 -14200.728} C_VEL
LIN {X 0,Y 340.777,Z 388.645,A -85,B 0,C 180,E1 -14204.449,E2 -14204.449} C_VEL
LIN {X 0,Y 340.832,Z 388.656,A -85,B 0,C 180,E1 -14208.1,E2 -14208.1} C_VEL
LIN {X 0,Y 340.965,Z 388.628,A -85,B 0,C 180,E1 -14211.704,E2 -14211.704} C_VEL
LIN {X 0,Y 340.994,Z 388.628,A -85,B 0,C 180,E1 -14214.085,E2 -14214.085} C_VEL
LIN {X 0,Y 341.113,Z 388.615,A -85,B 0,C 180,E1 -14217.639,E2 -14217.639} C_VEL
LIN {X 0,Y 341.096,Z 388.601,A -85,B 0,C 180,E1 -14221.181,E2 -14221.181} C_VEL
LIN {X 0,Y 341.111,Z 388.606,A -85,B 0,C 180,E1 -14222.362,E2 -14222.362} C_VEL
LIN {X 0,Y 341.004,Z 388.615,A -85,B 0,C 180,E1 -14227.103,E2 -14227.103} C_VEL
LIN {X 0,Y 340.831,Z 388.64,A -85,B 0,C 180,E1 -14230.695,E2 -14230.695} C_VEL
LIN {X 0,Y 340.849,Z 388.651,A -85,B 0,C 180,E1 -14234.326,E2 -14234.326} C_VEL
LIN {X 0,Y 340.771,Z 388.658,A -85,B 0,C 180,E1 -14238.441,E2 -14238.441} C_VEL
LIN {X 0,Y 340.704,Z 388.657,A -85,B 0,C 180,E1 -14241.843,E2 -14241.843} C_VEL
LIN {X 0,Y 340.657,Z 388.663,A -85,B 0,C 180,E1 -14245.674,E2 -14245.674} C_VEL
LIN {X 0,Y 340.662,Z 388.671,A -85,B 0,C 180,E1 -14248.327,E2 -14248.327} C_VEL
LIN {X 0,Y 340.67,Z 388.679,A -85,B 0,C 180,E1 -14251.048,E2 -14251.048} C_VEL
LIN {X 0,Y 340.703,Z 388.664,A -85,B 0,C 180,E1 -14255.281,E2 -14255.281} C_VEL
LIN {X 0,Y 340.681,Z 388.641,A -85,B 0,C 180,E1 -14258.384,E2 -14258.384} C_VEL
LIN {X 0,Y 340.679,Z 388.645,A -85,B 0,C 180,E1 -14262.045,E2 -14262.045} C_VEL
LIN {X 0,Y 340.692,Z 388.903,A -85,B 0,C 180,E1 -14263.095,E2 -14263.095} C_VEL
LIN {X 0,Y 346.066,Z 402.224,A -85,B 0,C 180,E1 -14266.068,E2 -14266.068} C_VEL
LIN {X 0,Y 351.194,Z 416.572,A -85,B 0,C 180,E1 -14268.971,E2 -14268.971} C_VEL
LIN {X 0,Y 355.458,Z 430.619,A -85,B 0,C 180,E1 -14271.597,E2 -14271.597} C_VEL
LIN {X 0,Y 358.394,Z 441.614,A -85,B 0,C 180,E1 -14273.514,E2 -14273.514} C_VEL
LIN {X 0,Y 356.605,Z 462.432,A -85,B 0,C 180,E1 -14276.216,E2 -14276.216} C_VEL
LIN {X 0,Y 355.869,Z 471.315,A -85,B 0,C 180,E1 -14277.282,E2 -14277.282} C_VEL
LIN {X 0,Y 360.922,Z 503.322,A -85,B 0,C 180,E1 -14278.541,E2 -14278.541} C_VEL
LIN {X 0,Y 361.854,Z 510.441,A -85,B 0,C 180,E1 -14278.793,E2 -14278.793} C_VEL
LIN {X 0,Y 358.058,Z 640.427,A -85,B 0,C 180,E1 -14281.419,E2 -14281.419} C_VEL
LIN {X 0,Y 357.169,Z 655.282,A -85,B 0,C 180,E1 -14281.91,E2 -14281.91} C_VEL
LIN {X 0,Y 355.829,Z 670.288,A -85,B 0,C 180,E1 -14282.626,E2 -14282.626} C_VEL
LIN {X 0,Y 354.214,Z 684.82,A -85,B 0,C 180,E1 -14283.563,E2 -14283.563} C_VEL
LIN {X 0,Y 352.553,Z 697.753,A -85,B 0,C 180,E1 -14284.624,E2 -14284.624} C_VEL
LIN {X 0,Y 350.41,Z 711.713,A -85,B 0,C 180,E1 -14286.039,E2 -14286.039} C_VEL
LIN {X 0,Y 348.343,Z 724.404,A -85,B 0,C 180,E1 -14287.634,E2 -14287.634} C_VEL
LIN {X 0,Y 346.533,Z 735.227,A -85,B 0,C 180,E1 -14289.281,E2 -14289.281} C_VEL
LIN {X 0,Y 344.497,Z 746.082,A -85,B 0,C 180,E1 -14291.26,E2 -14291.26} C_VEL
LIN {X 0,Y 342.868,Z 755.389,A -85,B 0,C 180,E1 -14293.326,E2 -14293.326} C_VEL
LIN {X 0,Y 341.705,Z 762.335,A -85,B 0,C 180,E1 -14295.166,E2 -14295.166} C_VEL
LIN {X 0,Y 340.638,Z 769.556,A -85,B 0,C 180,E1 -14297.491,E2 -14297.491} C_VEL
LIN {X 0,Y 339.787,Z 775.45,A -85,B 0,C 180,E1 -14299.876,E2 -14299.876} C_VEL
LIN {X 0,Y 339.422,Z 778.927,A -85,B 0,C 180,E1 -14301.668,E2 -14301.668} C_VEL
LIN {X 0,Y 339.086,Z 782.634,A -85,B 0,C 180,E1 -14304.191,E2 -14304.191} C_VEL
LIN {X 0,Y 339.034,Z 784.811,A -85,B 0,C 180,E1 -14306.436,E2 -14306.436} C_VEL
LIN {X 0,Y 338.953,Z 786.002,A -85,B 0,C 180,E1 -14308.814,E2 -14308.814} C_VEL
LIN {X 0,Y 338.953,Z 786.017,A -85,B 0,C 180,E1 -14311.19,E2 -14311.19} C_VEL
LIN {X 0,Y 339.037,Z 784.88,A -85,B 0,C 180,E1 -14313.567,E2 -14313.567} C_VEL
LIN {X 0,Y 339.134,Z 782.593,A -85,B 0,C 180,E1 -14315.949,E2 -14315.949} C_VEL
LIN {X 0,Y 339.433,Z 779.1,A -85,B 0,C 180,E1 -14318.335,E2 -14318.335} C_VEL
LIN {X 0,Y 339.908,Z 774.321,A -85,B 0,C 180,E1 -14320.726,E2 -14320.726} C_VEL
LIN {X 0,Y 340.869,Z 768.136,A -85,B 0,C 180,E1 -14323.11,E2 -14323.11} C_VEL
LIN {X 0,Y 342.03,Z 760.355,A -85,B 0,C 180,E1 -14325.495,E2 -14325.495} C_VEL
LIN {X 0,Y 343.464,Z 752.055,A -85,B 0,C 180,E1 -14327.568,E2 -14327.568} C_VEL
LIN {X 0,Y 344.981,Z 743.63,A -85,B 0,C 180,E1 -14329.334,E2 -14329.334} C_VEL
LIN {X 0,Y 346.996,Z 732.343,A -85,B 0,C 180,E1 -14331.302,E2 -14331.302} C_VEL
LIN {X 0,Y 348.097,Z 725.756,A -85,B 0,C 180,E1 -14332.286,E2 -14332.286} C_VEL
LIN {X 0,Y 348.218,Z 721.351,A -85,B 0,C 180,E1 -14332.934,E2 -14332.934} C_VEL
LIN {X 0,Y 345.558,Z 708.184,A -85,B 0,C 180,E1 -14334.881,E2 -14334.881} C_VEL
LIN {X 0,Y 345.379,Z 703.382,A -85,B 0,C 180,E1 -14335.448,E2 -14335.448} C_VEL
LIN {X 0,Y 345.562,Z 701.703,A -85,B 0,C 180,E1 -14335.615,E2 -14335.615} C_VEL
LIN {X 0,Y 347.699,Z 687.028,A -85,B 0,C 180,E1 -14336.891,E2 -14336.891} C_VEL
LIN {X 0,Y 349.33,Z 672.444,A -85,B 0,C 180,E1 -14337.89,E2 -14337.89} C_VEL
LIN {X 0,Y 350.725,Z 658.097,A -85,B 0,C 180,E1 -14338.625,E2 -14338.625} C_VEL
LIN {X 0,Y 351.801,Z 642.438,A -85,B 0,C 180,E1 -14339.182,E2 -14339.182} C_VEL
LIN {X 0,Y 353.149,Z 601.759,A -85,B 0,C 180,E1 -14340.044,E2 -14340.044} C_VEL
LIN {X 0,Y 355.79,Z 510.706,A -85,B 0,C 180,E1 -14341.9,E2 -14341.9} C_VEL
LIN {X 0,Y 350.732,Z 477.452,A -85,B 0,C 180,E1 -14343.207,E2 -14343.207} C_VEL
LIN {X 0,Y 349.713,Z 471.131,A -85,B 0,C 180,E1 -14343.489,E2 -14343.489} C_VEL
LIN {X 0,Y 351.598,Z 450.22,A -85,B 0,C 180,E1 -14346.135,E2 -14346.135} C_VEL
LIN {X 0,Y 352.105,Z 445.226,A -85,B 0,C 180,E1 -14346.786,E2 -14346.786} C_VEL
LIN {X 0,Y 351.241,Z 440.939,A -85,B 0,C 180,E1 -14347.508,E2 -14347.508} C_VEL
LIN {X 0,Y 346.814,Z 425.015,A -85,B 0,C 180,E1 -14350.427,E2 -14350.427} C_VEL
LIN {X 0,Y 342.143,Z 411.082,A -85,B 0,C 180,E1 -14353.23,E2 -14353.23} C_VEL
LIN {X 0,Y 336.363,Z 396.451,A -85,B 0,C 180,E1 -14356.409,E2 -14356.409} C_VEL
LIN {X 0,Y 333.694,Z 389.88,A -85,B 0,C 180,E1 -14357.983,E2 -14357.983} C_VEL
LIN {X 0,Y 333.621,Z 389.544,A -85,B 0,C 180,E1 -14358.427,E2 -14358.427} C_VEL
LIN {X 0,Y 333.647,Z 389.551,A -85,B 0,C 180,E1 -14362.348,E2 -14362.348} C_VEL
LIN {X 0,Y 333.678,Z 389.508,A -85,B 0,C 180,E1 -14365.342,E2 -14365.342} C_VEL
LIN {X 0,Y 333.626,Z 389.553,A -85,B 0,C 180,E1 -14368.221,E2 -14368.221} C_VEL
LIN {X 0,Y 333.695,Z 389.749,A -85,B 0,C 180,E1 -14371.609,E2 -14371.609} C_VEL
LIN {X 0,Y 334.471,Z 392.978,A -85,B 0,C 180,E1 -14372.368,E2 -14372.368} C_VEL
LIN {X 0,Y 345.994,Z 423.3,A -85,B 0,C 180,E1 -14374.058,E2 -14374.058} C_VEL
LIN {X 0,Y 341.955,Z 537.441,A -85,B 0,C 180,E1 -14377.304,E2 -14377.304} C_VEL
LIN {X 0,Y 341.493,Z 553.185,A -85,B 0,C 180,E1 -14378.01,E2 -14378.01} C_VEL
LIN {X 0,Y 340.743,Z 568.157,A -85,B 0,C 180,E1 -14378.921,E2 -14378.921} C_VEL
LIN {X 0,Y 339.82,Z 582.5,A -85,B 0,C 180,E1 -14380.047,E2 -14380.047} C_VEL
LIN {X 0,Y 338.892,Z 596.207,A -85,B 0,C 180,E1 -14381.407,E2 -14381.407} C_VEL
LIN {X 0,Y 337.874,Z 608.688,A -85,B 0,C 180,E1 -14382.914,E2 -14382.914} C_VEL
LIN {X 0,Y 336.998,Z 620.105,A -85,B 0,C 180,E1 -14384.58,E2 -14384.58} C_VEL
LIN {X 0,Y 336.081,Z 630.465,A -85,B 0,C 180,E1 -14386.393,E2 -14386.393} C_VEL
LIN {X 0,Y 335.439,Z 639.094,A -85,B 0,C 180,E1 -14388.213,E2 -14388.213} C_VEL
LIN {X 0,Y 334.796,Z 647.378,A -85,B 0,C 180,E1 -14390.332,E2 -14390.332} C_VEL
LIN {X 0,Y 334.493,Z 653.24,A -85,B 0,C 180,E1 -14392.15,E2 -14392.15} C_VEL
LIN {X 0,Y 334.125,Z 658.03,A -85,B 0,C 180,E1 -14393.963,E2 -14393.963} C_VEL
LIN {X 0,Y 333.874,Z 661.883,A -85,B 0,C 180,E1 -14395.775,E2 -14395.775} C_VEL
LIN {X 0,Y 333.919,Z 664.864,A -85,B 0,C 180,E1 -14397.587,E2 -14397.587} C_VEL
LIN {X 0,Y 333.995,Z 667.518,A -85,B 0,C 180,E1 -14400,E2 -14400} C_VEL
LIN {X 0,Y 334.532,Z 668.716,A -85,B 0,C 180,E1 -14402.408,E2 -14402.408} C_VEL
LIN {X 0,Y 335.164,Z 668.515,A -85,B 0,C 180,E1 -14404.811,E2 -14404.811} C_VEL
LIN {X 0,Y 335.953,Z 666.912,A -85,B 0,C 180,E1 -14407.211,E2 -14407.211} C_VEL
LIN {X 0,Y 337.203,Z 663.835,A -85,B 0,C 180,E1 -14409.598,E2 -14409.598} C_VEL
LIN {X 0,Y 338.335,Z 660.451,A -85,B 0,C 180,E1 -14411.381,E2 -14411.381} C_VEL
LIN {X 0,Y 339.632,Z 656.165,A -85,B 0,C 180,E1 -14413.157,E2 -14413.157} C_VEL
LIN {X 0,Y 341.39,Z 649.918,A -85,B 0,C 180,E1 -14415.217,E2 -14415.217} C_VEL
LIN {X 0,Y 343.407,Z 642.069,A -85,B 0,C 180,E1 -14417.262,E2 -14417.262} C_VEL
LIN {X 0,Y 345.349,Z 633.909,A -85,B 0,C 180,E1 -14419.002,E2 -14419.002} C_VEL
LIN {X 0,Y 347.512,Z 624.181,A -85,B 0,C 180,E1 -14420.713,E2 -14420.713} C_VEL
LIN {X 0,Y 349.863,Z 612.17,A -85,B 0,C 180,E1 -14422.437,E2 -14422.437} C_VEL
LIN {X 0,Y 351.914,Z 600.197,A -85,B 0,C 180,E1 -14423.854,E2 -14423.854} C_VEL
LIN {X 0,Y 353.933,Z 586.95,A -85,B 0,C 180,E1 -14425.115,E2 -14425.115} C_VEL
LIN {X 0,Y 355.775,Z 572.501,A -85,B 0,C 180,E1 -14426.231,E2 -14426.231} C_VEL
LIN {X 0,Y 357.378,Z 556.435,A -85,B 0,C 180,E1 -14427.172,E2 -14427.172} C_VEL
LIN {X 0,Y 358.936,Z 537.406,A -85,B 0,C 180,E1 -14427.999,E2 -14427.999} C_VEL
LIN {X 0,Y 365.461,Z 482.172,A -85,B 0,C 180,E1 -14430.082,E2 -14430.082} C_VEL
LIN {X 0,Y 369.696,Z 450.587,A -85,B 0,C 180,E1 -14431.257,E2 -14431.257} C_VEL
LIN {X 0,Y 365.893,Z 444.373,A -85,B 0,C 180,E1 -14432.735,E2 -14432.735} C_VEL
LIN {X 0,Y 362.366,Z 439.275,A -85,B 0,C 180,E1 -14434.321,E2 -14434.321} C_VEL
LIN {X 0,Y 359.446,Z 435.875,A -85,B 0,C 180,E1 -14435.847,E2 -14435.847} C_VEL
LIN {X 0,Y 356.813,Z 432.961,A -85,B 0,C 180,E1 -14437.632,E2 -14437.632} C_VEL
LIN {X 0,Y 354.287,Z 430.838,A -85,B 0,C 180,E1 -14440.246,E2 -14440.246} C_VEL
LIN {X 0,Y 353.28,Z 431.252,A -85,B 0,C 180,E1 -14442.601,E2 -14442.601} C_VEL
LIN {X 0,Y 353.57,Z 432.807,A -85,B 0,C 180,E1 -14444.719,E2 -14444.719} C_VEL
LIN {X 0,Y 354.764,Z 435.757,A -85,B 0,C 180,E1 -14446.738,E2 -14446.738} C_VEL
LIN {X 0,Y 356.802,Z 440.07,A -85,B 0,C 180,E1 -14448.699,E2 -14448.699} C_VEL
LIN {X 0,Y 358.635,Z 443.939,A -85,B 0,C 180,E1 -14449.993,E2 -14449.993} C_VEL
LIN {X 0,Y 362.042,Z 451.976,A -85,B 0,C 180,E1 -14451.969,E2 -14451.969} C_VEL
LIN {X 0,Y 362.838,Z 454.578,A -85,B 0,C 180,E1 -14452.42,E2 -14452.42} C_VEL
LIN {X 0,Y 363.689,Z 467.245,A -85,B 0,C 180,E1 -14453.59,E2 -14453.59} C_VEL
LIN {X 0,Y 364.47,Z 483.434,A -85,B 0,C 180,E1 -14454.846,E2 -14454.846} C_VEL
LIN {X 0,Y 364.708,Z 498.212,A -85,B 0,C 180,E1 -14455.783,E2 -14455.783} C_VEL
LIN {X 0,Y 364.436,Z 510.811,A -85,B 0,C 180,E1 -14456.434,E2 -14456.434} C_VEL
LIN {X 0,Y 357.955,Z 577.374,A -85,B 0,C 180,E1 -14458.646,E2 -14458.646} C_VEL
LIN {X 0,Y 354.896,Z 610.956,A -85,B 0,C 180,E1 -14459.751,E2 -14459.751} C_VEL
LIN {X 0,Y 352.601,Z 628.16,A -85,B 0,C 180,E1 -14460.522,E2 -14460.522} C_VEL
LIN {X 0,Y 351.56,Z 635.128,A -85,B 0,C 180,E1 -14460.878,E2 -14460.878} C_VEL
LIN {X 0,Y 350.671,Z 650.858,A -85,B 0,C 180,E1 -14461.33,E2 -14461.33} C_VEL
LIN {X 0,Y 349.521,Z 665.257,A -85,B 0,C 180,E1 -14461.963,E2 -14461.963} C_VEL
LIN {X 0,Y 348.072,Z 679.666,A -85,B 0,C 180,E1 -14462.832,E2 -14462.832} C_VEL
LIN {X 0,Y 346.201,Z 694.115,A -85,B 0,C 180,E1 -14463.959,E2 -14463.959} C_VEL
LIN {X 0,Y 344.225,Z 707.343,A -85,B 0,C 180,E1 -14465.256,E2 -14465.256} C_VEL
LIN {X 0,Y 342.169,Z 719.488,A -85,B 0,C 180,E1 -14466.708,E2 -14466.708} C_VEL
LIN {X 0,Y 340.118,Z 731.187,A -85,B 0,C 180,E1 -14468.412,E2 -14468.412} C_VEL
LIN {X 0,Y 338.219,Z 741.716,A -85,B 0,C 180,E1 -14470.264,E2 -14470.264} C_VEL
LIN {X 0,Y 336.394,Z 751.598,A -85,B 0,C 180,E1 -14472.364,E2 -14472.364} C_VEL
LIN {X 0,Y 334.932,Z 759.785,A -85,B 0,C 180,E1 -14474.478,E2 -14474.478} C_VEL
LIN {X 0,Y 333.872,Z 766.564,A -85,B 0,C 180,E1 -14476.61,E2 -14476.61} C_VEL
LIN {X 0,Y 332.913,Z 772.828,A -85,B 0,C 180,E1 -14479.046,E2 -14479.046} C_VEL
LIN {X 0,Y 332.424,Z 777.667,A -85,B 0,C 180,E1 -14481.488,E2 -14481.488} C_VEL
LIN {X 0,Y 332.136,Z 781.295,A -85,B 0,C 180,E1 -14483.998,E2 -14483.998} C_VEL
LIN {X 0,Y 332.035,Z 783.534,A -85,B 0,C 180,E1 -14486.357,E2 -14486.357} C_VEL
LIN {X 0,Y 331.937,Z 784.701,A -85,B 0,C 180,E1 -14488.785,E2 -14488.785} C_VEL
LIN {X 0,Y 331.94,Z 784.698,A -85,B 0,C 180,E1 -14491.211,E2 -14491.211} C_VEL
LIN {X 0,Y 332.036,Z 783.523,A -85,B 0,C 180,E1 -14493.639,E2 -14493.639} C_VEL
LIN {X 0,Y 332.12,Z 781.192,A -85,B 0,C 180,E1 -14496.072,E2 -14496.072} C_VEL
LIN {X 0,Y 332.419,Z 777.65,A -85,B 0,C 180,E1 -14498.509,E2 -14498.509} C_VEL
LIN {X 0,Y 332.905,Z 772.807,A -85,B 0,C 180,E1 -14500.951,E2 -14500.951} C_VEL
LIN {X 0,Y 333.858,Z 766.529,A -85,B 0,C 180,E1 -14503.387,E2 -14503.387} C_VEL
LIN {X 0,Y 335.112,Z 758.638,A -85,B 0,C 180,E1 -14505.819,E2 -14505.819} C_VEL
LIN {X 0,Y 336.58,Z 750.211,A -85,B 0,C 180,E1 -14507.936,E2 -14507.936} C_VEL
LIN {X 0,Y 338.188,Z 741.657,A -85,B 0,C 180,E1 -14509.734,E2 -14509.734} C_VEL
LIN {X 0,Y 339.935,Z 731.605,A -85,B 0,C 180,E1 -14511.51,E2 -14511.51} C_VEL
LIN {X 0,Y 342.153,Z 719.412,A -85,B 0,C 180,E1 -14513.289,E2 -14513.289} C_VEL
LIN {X 0,Y 344.38,Z 705.898,A -85,B 0,C 180,E1 -14514.89,E2 -14514.89} C_VEL
LIN {X 0,Y 346.362,Z 692.321,A -85,B 0,C 180,E1 -14516.186,E2 -14516.186} C_VEL
LIN {X 0,Y 348.044,Z 678.894,A -85,B 0,C 180,E1 -14517.214,E2 -14517.214} C_VEL
LIN {X 0,Y 349.619,Z 663.651,A -85,B 0,C 180,E1 -14518.106,E2 -14518.106} C_VEL
LIN {X 0,Y 350.797,Z 648.599,A -85,B 0,C 180,E1 -14518.737,E2 -14518.737} C_VEL
LIN {X 0,Y 351.577,Z 632.917,A -85,B 0,C 180,E1 -14519.158,E2 -14519.158} C_VEL
LIN {X 0,Y 354.813,Z 520.82,A -85,B 0,C 180,E1 -14521.431,E2 -14521.431} C_VEL
LIN {X 0,Y 355.014,Z 506.146,A -85,B 0,C 180,E1 -14521.752,E2 -14521.752} C_VEL
LIN {X 0,Y 351.212,Z 474.901,A -85,B 0,C 180,E1 -14522.879,E2 -14522.879} C_VEL
LIN {X 0,Y 350.086,Z 466.575,A -85,B 0,C 180,E1 -14523.202,E2 -14523.202} C_VEL
LIN {X 0,Y 348.755,Z 438.377,A -85,B 0,C 180,E1 -14525.12,E2 -14525.12} C_VEL
LIN {X 0,Y 348.254,Z 435.881,A -85,B 0,C 180,E1 -14525.329,E2 -14525.329} C_VEL
LIN {X 0,Y 342.422,Z 420.006,A -85,B 0,C 180,E1 -14527.072,E2 -14527.072} C_VEL
LIN {X 0,Y 336.964,Z 400.992,A -85,B 0,C 180,E1 -14530.596,E2 -14530.596} C_VEL
LIN {X 0,Y 333.692,Z 389.703,A -85,B 0,C 180,E1 -14532.877,E2 -14532.877} C_VEL
LIN {X 0,Y 333.614,Z 389.508,A -85,B 0,C 180,E1 -14537.5,E2 -14537.5} C_VEL
LIN {X 0,Y 333.621,Z 389.553,A -85,B 0,C 180,E1 -14541.205,E2 -14541.205} C_VEL
LIN {X 0,Y 333.66,Z 389.496,A -85,B 0,C 180,E1 -14543.859,E2 -14543.859} C_VEL
LIN {X 0,Y 333.63,Z 389.536,A -85,B 0,C 180,E1 -14547.412,E2 -14547.412} C_VEL
LIN {X 0,Y 333.619,Z 389.538,A -85,B 0,C 180,E1 -14551.019,E2 -14551.019} C_VEL
LIN {X 0,Y 333.619,Z 389.55,A -85,B 0,C 180,E1 -14553.744,E2 -14553.744} C_VEL
LIN {X 0,Y 333.628,Z 389.541,A -85,B 0,C 180,E1 -14556.407,E2 -14556.407} C_VEL
LIN {X 0,Y 333.639,Z 389.539,A -85,B 0,C 180,E1 -14559.017,E2 -14559.017} C_VEL
LIN {X 0,Y 333.698,Z 389.539,A -85,B 0,C 180,E1 -14561.584,E2 -14561.584} C_VEL
LIN {X 0,Y 333.759,Z 389.517,A -85,B 0,C 180,E1 -14565.6,E2 -14565.6} C_VEL
LIN {X 0,Y 333.8,Z 389.521,A -85,B 0,C 180,E1 -14569.077,E2 -14569.077} C_VEL
LIN {X 0,Y 333.938,Z 389.513,A -85,B 0,C 180,E1 -14572.746,E2 -14572.746} C_VEL
LIN {X 0,Y 333.766,Z 389.514,A -85,B 0,C 180,E1 -14575.169,E2 -14575.169} C_VEL
LIN {X 0,Y 334.053,Z 389.495,A -85,B 0,C 180,E1 -14577.589,E2 -14577.589} C_VEL
LIN {X 0,Y 334.064,Z 389.476,A -85,B 0,C 180,E1 -14581.206,E2 -14581.206} C_VEL
LIN {X 0,Y 333.791,Z 389.531,A -85,B 0,C 180,E1 -14583.622,E2 -14583.622} C_VEL
LIN {X 0,Y 333.95,Z 389.492,A -85,B 0,C 180,E1 -14586.711,E2 -14586.711} C_VEL
LIN {X 0,Y 333.805,Z 389.527,A -85,B 0,C 180,E1 -14589.697,E2 -14589.697} C_VEL
LIN {X 0,Y 333.782,Z 389.527,A -85,B 0,C 180,E1 -14593.392,E2 -14593.392} C_VEL
LIN {X 0,Y 333.704,Z 389.525,A -85,B 0,C 180,E1 -14597.149,E2 -14597.149} C_VEL
LIN {X 0,Y 333.656,Z 389.545,A -85,B 0,C 180,E1 -14599.695,E2 -14599.695} C_VEL
LIN {X 0,Y 333.628,Z 389.551,A -85,B 0,C 180,E1 -14603.593,E2 -14603.593} C_VEL
LIN {X 0,Y 333.615,Z 389.544,A -85,B 0,C 180,E1 -14606.257,E2 -14606.257} C_VEL
LIN {X 0,Y 333.615,Z 389.543,A -85,B 0,C 180,E1 -14608.981,E2 -14608.981} C_VEL
LIN {X 0,Y 333.627,Z 389.545,A -85,B 0,C 180,E1 -14612.587,E2 -14612.587} C_VEL
LIN {X 0,Y 333.661,Z 389.52,A -85,B 0,C 180,E1 -14616.141,E2 -14616.141} C_VEL
LIN {X 0,Y 333.59,Z 389.537,A -85,B 0,C 180,E1 -14619.2,E2 -14619.2} C_VEL
LIN {X 0,Y 333.676,Z 389.7,A -85,B 0,C 180,E1 -14622.071,E2 -14622.071} C_VEL
LIN {X 0,Y 334.413,Z 391.967,A -85,B 0,C 180,E1 -14622.649,E2 -14622.649} C_VEL
LIN {X 0,Y 339.127,Z 403.158,A -85,B 0,C 180,E1 -14625.205,E2 -14625.205} C_VEL
LIN {X 0,Y 344.306,Z 417.265,A -85,B 0,C 180,E1 -14628.163,E2 -14628.163} C_VEL
LIN {X 0,Y 348.87,Z 432.214,A -85,B 0,C 180,E1 -14631.035,E2 -14631.035} C_VEL
LIN {X 0,Y 351.893,Z 443.344,A -85,B 0,C 180,E1 -14633.023,E2 -14633.023} C_VEL
LIN {X 0,Y 352,Z 445.753,A -85,B 0,C 180,E1 -14633.384,E2 -14633.384} C_VEL
LIN {X 0,Y 349.983,Z 467.137,A -85,B 0,C 180,E1 -14636.137,E2 -14636.137} C_VEL
LIN {X 0,Y 349.694,Z 471.493,A -85,B 0,C 180,E1 -14636.643,E2 -14636.643} C_VEL
LIN {X 0,Y 354.806,Z 503.931,A -85,B 0,C 180,E1 -14637.952,E2 -14637.952} C_VEL
LIN {X 0,Y 355.754,Z 512.307,A -85,B 0,C 180,E1 -14638.242,E2 -14638.242} C_VEL
LIN {X 0,Y 351.853,Z 640.346,A -85,B 0,C 180,E1 -14640.867,E2 -14640.867} C_VEL
LIN {X 0,Y 350.935,Z 655.231,A -85,B 0,C 180,E1 -14641.365,E2 -14641.365} C_VEL
LIN {X 0,Y 349.53,Z 670.251,A -85,B 0,C 180,E1 -14642.091,E2 -14642.091} C_VEL
LIN {X 0,Y 347.792,Z 685.326,A -85,B 0,C 180,E1 -14643.081,E2 -14643.081} C_VEL
LIN {X 0,Y 345.91,Z 699.272,A -85,B 0,C 180,E1 -14644.263,E2 -14644.263} C_VEL
LIN {X 0,Y 343.883,Z 711.691,A -85,B 0,C 180,E1 -14645.555,E2 -14645.555} C_VEL
LIN {X 0,Y 341.763,Z 724.279,A -85,B 0,C 180,E1 -14647.163,E2 -14647.163} C_VEL
LIN {X 0,Y 339.81,Z 735.519,A -85,B 0,C 180,E1 -14648.908,E2 -14648.908} C_VEL
LIN {X 0,Y 337.707,Z 746.066,A -85,B 0,C 180,E1 -14650.869,E2 -14650.869} C_VEL
LIN {X 0,Y 336.031,Z 755.374,A -85,B 0,C 180,E1 -14652.976,E2 -14652.976} C_VEL
LIN {X 0,Y 334.713,Z 762.764,A -85,B 0,C 180,E1 -14654.987,E2 -14654.987} C_VEL
LIN {X 0,Y 333.653,Z 769.542,A -85,B 0,C 180,E1 -14657.224,E2 -14657.224} C_VEL
LIN {X 0,Y 332.75,Z 775.436,A -85,B 0,C 180,E1 -14659.66,E2 -14659.66} C_VEL
LIN {X 0,Y 332.355,Z 778.913,A -85,B 0,C 180,E1 -14661.49,E2 -14661.49} C_VEL
LIN {X 0,Y 332.012,Z 782.787,A -85,B 0,C 180,E1 -14664.207,E2 -14664.207} C_VEL
LIN {X 0,Y 331.939,Z 784.797,A -85,B 0,C 180,E1 -14666.36,E2 -14666.36} C_VEL
LIN {X 0,Y 331.861,Z 785.989,A -85,B 0,C 180,E1 -14668.788,E2 -14668.788} C_VEL
LIN {X 0,Y 331.862,Z 786.003,A -85,B 0,C 180,E1 -14671.215,E2 -14671.215} C_VEL
LIN {X 0,Y 331.942,Z 784.866,A -85,B 0,C 180,E1 -14673.644,E2 -14673.644} C_VEL
LIN {X 0,Y 332.044,Z 782.578,A -85,B 0,C 180,E1 -14676.077,E2 -14676.077} C_VEL
LIN {X 0,Y 332.361,Z 779.084,A -85,B 0,C 180,E1 -14678.514,E2 -14678.514} C_VEL
LIN {X 0,Y 332.878,Z 774.305,A -85,B 0,C 180,E1 -14680.955,E2 -14680.955} C_VEL
LIN {X 0,Y 333.88,Z 768.118,A -85,B 0,C 180,E1 -14683.39,E2 -14683.39} C_VEL
LIN {X 0,Y 335.147,Z 760.336,A -85,B 0,C 180,E1 -14685.821,E2 -14685.821} C_VEL
LIN {X 0,Y 336.654,Z 752.034,A -85,B 0,C 180,E1 -14687.936,E2 -14687.936} C_VEL
LIN {X 0,Y 338.256,Z 743.609,A -85,B 0,C 180,E1 -14689.734,E2 -14689.734} C_VEL
LIN {X 0,Y 340.224,Z 732.969,A -85,B 0,C 180,E1 -14691.633,E2 -14691.633} C_VEL
LIN {X 0,Y 342.408,Z 720.731,A -85,B 0,C 180,E1 -14693.435,E2 -14693.435} C_VEL
LIN {X 0,Y 344.414,Z 708.698,A -85,B 0,C 180,E1 -14694.891,E2 -14694.891} C_VEL
LIN {X 0,Y 345.562,Z 701.703,A -85,B 0,C 180,E1 -14695.615,E2 -14695.615} C_VEL
LIN {X 0,Y 345.823,Z 696.659,A -85,B 0,C 180,E1 -14696.129,E2 -14696.129} C_VEL
LIN {X 0,Y 344.421,Z 688.488,A -85,B 0,C 180,E1 -14697.036,E2 -14697.036} C_VEL
LIN {X 0,Y 342.854,Z 680.122,A -85,B 0,C 180,E1 -14697.886,E2 -14697.886} C_VEL
LIN {X 0,Y 342.814,Z 674.773,A -85,B 0,C 180,E1 -14698.297,E2 -14698.297} C_VEL
LIN {X 0,Y 344.3,Z 660.317,A -85,B 0,C 180,E1 -14699.084,E2 -14699.084} C_VEL
LIN {X 0,Y 345.493,Z 644.72,A -85,B 0,C 180,E1 -14699.685,E2 -14699.685} C_VEL
LIN {X 0,Y 346.28,Z 624.79,A -85,B 0,C 180,E1 -14700.155,E2 -14700.155} C_VEL
LIN {X 0,Y 349.771,Z 512.164,A -85,B 0,C 180,E1 -14702.477,E2 -14702.477} C_VEL
LIN {X 0,Y 345.34,Z 481.895,A -85,B 0,C 180,E1 -14703.682,E2 -14703.682} C_VEL
LIN {X 0,Y 343.596,Z 471.034,A -85,B 0,C 180,E1 -14704.166,E2 -14704.166} C_VEL
LIN {X 0,Y 345.703,Z 448.847,A -85,B 0,C 180,E1 -14707.012,E2 -14707.012} C_VEL
LIN {X 0,Y 345.795,Z 446.89,A -85,B 0,C 180,E1 -14707.286,E2 -14707.286} C_VEL
LIN {X 0,Y 341.704,Z 431.406,A -85,B 0,C 180,E1 -14710.123,E2 -14710.123} C_VEL
LIN {X 0,Y 337.269,Z 417.636,A -85,B 0,C 180,E1 -14712.88,E2 -14712.88} C_VEL
LIN {X 0,Y 332.303,Z 404.48,A -85,B 0,C 180,E1 -14715.739,E2 -14715.739} C_VEL
LIN {X 0,Y 327.74,Z 393.516,A -85,B 0,C 180,E1 -14718.336,E2 -14718.336} C_VEL
LIN {X 0,Y 326.606,Z 390.633,A -85,B 0,C 180,E1 -14719.098,E2 -14719.098} C_VEL
LIN {X 0,Y 326.63,Z 390.418,A -85,B 0,C 180,E1 -14722.953,E2 -14722.953} C_VEL
LIN {X 0,Y 326.61,Z 390.391,A -85,B 0,C 180,E1 -14725.981,E2 -14725.981} C_VEL
LIN {X 0,Y 326.614,Z 390.427,A -85,B 0,C 180,E1 -14729.399,E2 -14729.399} C_VEL
LIN {X 0,Y 326.672,Z 390.64,A -85,B 0,C 180,E1 -14731.225,E2 -14731.225} C_VEL
LIN {X 0,Y 327.374,Z 393.582,A -85,B 0,C 180,E1 -14731.906,E2 -14731.906} C_VEL
LIN {X 0,Y 339.365,Z 425.064,A -85,B 0,C 180,E1 -14733.709,E2 -14733.709} C_VEL
LIN {X 0,Y 335.119,Z 536.858,A -85,B 0,C 180,E1 -14736.982,E2 -14736.982} C_VEL
LIN {X 0,Y 334.599,Z 552.461,A -85,B 0,C 180,E1 -14737.672,E2 -14737.672} C_VEL
LIN {X 0,Y 333.847,Z 568.108,A -85,B 0,C 180,E1 -14738.626,E2 -14738.626} C_VEL
LIN {X 0,Y 332.904,Z 582.686,A -85,B 0,C 180,E1 -14739.776,E2 -14739.776} C_VEL
LIN {X 0,Y 331.97,Z 596.552,A -85,B 0,C 180,E1 -14741.164,E2 -14741.164} C_VEL
LIN {X 0,Y 330.925,Z 609.154,A -85,B 0,C 180,E1 -14742.703,E2 -14742.703} C_VEL
LIN {X 0,Y 330.102,Z 619.702,A -85,B 0,C 180,E1 -14744.249,E2 -14744.249} C_VEL
LIN {X 0,Y 329.112,Z 630.317,A -85,B 0,C 180,E1 -14746.099,E2 -14746.099} C_VEL
LIN {X 0,Y 328.467,Z 639.171,A -85,B 0,C 180,E1 -14747.959,E2 -14747.959} C_VEL
LIN {X 0,Y 327.796,Z 647.716,A -85,B 0,C 180,E1 -14750.124,E2 -14750.124} C_VEL
LIN {X 0,Y 327.457,Z 653.686,A -85,B 0,C 180,E1 -14751.981,E2 -14751.981} C_VEL
LIN {X 0,Y 327.093,Z 658.595,A -85,B 0,C 180,E1 -14753.833,E2 -14753.833} C_VEL
LIN {X 0,Y 326.833,Z 662.591,A -85,B 0,C 180,E1 -14755.684,E2 -14755.684} C_VEL
LIN {X 0,Y 326.894,Z 665.706,A -85,B 0,C 180,E1 -14757.535,E2 -14757.535} C_VEL
LIN {X 0,Y 326.953,Z 667.296,A -85,B 0,C 180,E1 -14758.768,E2 -14758.768} C_VEL
LIN {X 0,Y 326.968,Z 668.527,A -85,B 0,C 180,E1 -14760,E2 -14760} C_VEL
LIN {X 0,Y 327.542,Z 669.871,A -85,B 0,C 180,E1 -14762.459,E2 -14762.459} C_VEL
LIN {X 0,Y 328.21,Z 669.821,A -85,B 0,C 180,E1 -14764.913,E2 -14764.913} C_VEL
LIN {X 0,Y 329.069,Z 668.373,A -85,B 0,C 180,E1 -14767.362,E2 -14767.362} C_VEL
LIN {X 0,Y 330.386,Z 665.435,A -85,B 0,C 180,E1 -14769.798,E2 -14769.798} C_VEL
LIN {X 0,Y 332.066,Z 660.989,A -85,B 0,C 180,E1 -14772.219,E2 -14772.219} C_VEL
LIN {X 0,Y 333.917,Z 655.214,A -85,B 0,C 180,E1 -14774.491,E2 -14774.491} C_VEL
LIN {X 0,Y 336.02,Z 647.901,A -85,B 0,C 180,E1 -14776.713,E2 -14776.713} C_VEL
LIN {X 0,Y 338.336,Z 639.355,A -85,B 0,C 180,E1 -14778.782,E2 -14778.782} C_VEL
LIN {X 0,Y 340.611,Z 630.355,A -85,B 0,C 180,E1 -14780.534,E2 -14780.534} C_VEL
LIN {X 0,Y 342.915,Z 620.276,A -85,B 0,C 180,E1 -14782.186,E2 -14782.186} C_VEL
LIN {X 0,Y 345.141,Z 608.957,A -85,B 0,C 180,E1 -14783.713,E2 -14783.713} C_VEL
LIN {X 0,Y 347.393,Z 596.146,A -85,B 0,C 180,E1 -14785.141,E2 -14785.141} C_VEL
LIN {X 0,Y 349.669,Z 581.84,A -85,B 0,C 180,E1 -14786.403,E2 -14786.403} C_VEL
LIN {X 0,Y 351.428,Z 567.91,A -85,B 0,C 180,E1 -14787.385,E2 -14787.385} C_VEL
LIN {X 0,Y 352.887,Z 553.174,A -85,B 0,C 180,E1 -14788.193,E2 -14788.193} C_VEL
LIN {X 0,Y 354.754,Z 533.545,A -85,B 0,C 180,E1 -14789.026,E2 -14789.026} C_VEL
LIN {X 0,Y 362.578,Z 474.165,A -85,B 0,C 180,E1 -14791.313,E2 -14791.313} C_VEL
LIN {X 0,Y 365.4,Z 454.544,A -85,B 0,C 180,E1 -14792.066,E2 -14792.066} C_VEL
LIN {X 0,Y 362.431,Z 449.609,A -85,B 0,C 180,E1 -14793.332,E2 -14793.332} C_VEL
LIN {X 0,Y 359.435,Z 445.262,A -85,B 0,C 180,E1 -14794.791,E2 -14794.791} C_VEL
LIN {X 0,Y 357.002,Z 442.269,A -85,B 0,C 180,E1 -14796.181,E2 -14796.181} C_VEL
LIN {X 0,Y 354.765,Z 439.692,A -85,B 0,C 180,E1 -14797.797,E2 -14797.797} C_VEL
LIN {X 0,Y 352.678,Z 437.854,A -85,B 0,C 180,E1 -14799.974,E2 -14799.974} C_VEL
LIN {X 0,Y 351.673,Z 437.855,A -85,B 0,C 180,E1 -14801.819,E2 -14801.819} C_VEL
LIN {X 0,Y 351.536,Z 439.051,A -85,B 0,C 180,E1 -14803.967,E2 -14803.967} C_VEL
LIN {X 0,Y 352.286,Z 441.221,A -85,B 0,C 180,E1 -14805.8,E2 -14805.8} C_VEL
LIN {X 0,Y 353.853,Z 444.94,A -85,B 0,C 180,E1 -14807.743,E2 -14807.743} C_VEL
LIN {X 0,Y 355.861,Z 449.4,A -85,B 0,C 180,E1 -14809.401,E2 -14809.401} C_VEL
LIN {X 0,Y 359.006,Z 457.494,A -85,B 0,C 180,E1 -14811.445,E2 -14811.445} C_VEL
LIN {X 0,Y 359.4,Z 459.064,A -85,B 0,C 180,E1 -14811.716,E2 -14811.716} C_VEL
LIN {X 0,Y 359.964,Z 472.772,A -85,B 0,C 180,E1 -14812.987,E2 -14812.987} C_VEL
LIN {X 0,Y 360.364,Z 488.264,A -85,B 0,C 180,E1 -14814.19,E2 -14814.19} C_VEL
LIN {X 0,Y 360.305,Z 501.782,A -85,B 0,C 180,E1 -14815.048,E2 -14815.048} C_VEL
LIN {X 0,Y 359.862,Z 512.621,A -85,B 0,C 180,E1 -14815.614,E2 -14815.614} C_VEL
LIN {X 0,Y 352.726,Z 580.208,A -85,B 0,C 180,E1 -14817.917,E2 -14817.917} C_VEL
LIN {X 0,Y 349.779,Z 609.684,A -85,B 0,C 180,E1 -14818.925,E2 -14818.925} C_VEL
LIN {X 0,Y 347.386,Z 626.607,A -85,B 0,C 180,E1 -14819.699,E2 -14819.699} C_VEL
LIN {X 0,Y 345.167,Z 639.614,A -85,B 0,C 180,E1 -14820.41,E2 -14820.41} C_VEL
LIN {X 0,Y 344.213,Z 654.524,A -85,B 0,C 180,E1 -14820.908,E2 -14820.908} C_VEL
LIN {X 0,Y 342.87,Z 669.162,A -85,B 0,C 180,E1 -14821.62,E2 -14821.62} C_VEL
LIN {X 0,Y 341.331,Z 683.511,A -85,B 0,C 180,E1 -14822.571,E2 -14822.571} C_VEL
LIN {X 0,Y 339.366,Z 697.286,A -85,B 0,C 180,E1 -14823.725,E2 -14823.725} C_VEL
LIN {X 0,Y 337.332,Z 709.936,A -85,B 0,C 180,E1 -14825.044,E2 -14825.044} C_VEL
LIN {X 0,Y 335.044,Z 722.704,A -85,B 0,C 180,E1 -14826.674,E2 -14826.674} C_VEL
LIN {X 0,Y 333.048,Z 733.488,A -85,B 0,C 180,E1 -14828.348,E2 -14828.348} C_VEL
LIN {X 0,Y 331.175,Z 743.228,A -85,B 0,C 180,E1 -14830.149,E2 -14830.149} C_VEL
LIN {X 0,Y 329.351,Z 752.849,A -85,B 0,C 180,E1 -14832.295,E2 -14832.295} C_VEL
LIN {X 0,Y 327.85,Z 760.855,A -85,B 0,C 180,E1 -14834.456,E2 -14834.456} C_VEL
LIN {X 0,Y 326.648,Z 768.297,A -85,B 0,C 180,E1 -14836.942,E2 -14836.942} C_VEL
LIN {X 0,Y 325.739,Z 774.196,A -85,B 0,C 180,E1 -14839.431,E2 -14839.431} C_VEL
LIN {X 0,Y 325.356,Z 777.682,A -85,B 0,C 180,E1 -14841.301,E2 -14841.301} C_VEL
LIN {X 0,Y 325.03,Z 781.539,A -85,B 0,C 180,E1 -14844.064,E2 -14844.064} C_VEL
LIN {X 0,Y 324.939,Z 783.548,A -85,B 0,C 180,E1 -14846.278,E2 -14846.278} C_VEL
LIN {X 0,Y 324.846,Z 784.714,A -85,B 0,C 180,E1 -14848.758,E2 -14848.758} C_VEL
LIN {X 0,Y 324.849,Z 784.712,A -85,B 0,C 180,E1 -14851.238,E2 -14851.238} C_VEL
LIN {X 0,Y 324.939,Z 783.537,A -85,B 0,C 180,E1 -14853.718,E2 -14853.718} C_VEL
LIN {X 0,Y 325.044,Z 781.205,A -85,B 0,C 180,E1 -14856.204,E2 -14856.204} C_VEL
LIN {X 0,Y 325.351,Z 777.664,A -85,B 0,C 180,E1 -14858.695,E2 -14858.695} C_VEL
LIN {X 0,Y 325.884,Z 772.821,A -85,B 0,C 180,E1 -14861.19,E2 -14861.19} C_VEL
LIN {X 0,Y 326.871,Z 766.544,A -85,B 0,C 180,E1 -14863.678,E2 -14863.678} C_VEL
LIN {X 0,Y 328.231,Z 758.653,A -85,B 0,C 180,E1 -14866.16,E2 -14866.16} C_VEL
LIN {X 0,Y 329.796,Z 750.227,A -85,B 0,C 180,E1 -14868.318,E2 -14868.318} C_VEL
LIN {X 0,Y 331.49,Z 741.674,A -85,B 0,C 180,E1 -14870.15,E2 -14870.15} C_VEL
LIN {X 0,Y 333.454,Z 730.971,A -85,B 0,C 180,E1 -14872.067,E2 -14872.067} C_VEL
LIN {X 0,Y 335.597,Z 719.432,A -85,B 0,C 180,E1 -14873.772,E2 -14873.772} C_VEL
LIN {X 0,Y 337.93,Z 705.921,A -85,B 0,C 180,E1 -14875.398,E2 -14875.398} C_VEL
LIN {X 0,Y 339.983,Z 692.349,A -85,B 0,C 180,E1 -14876.716,E2 -14876.716} C_VEL
LIN {X 0,Y 341.824,Z 678.424,A -85,B 0,C 180,E1 -14877.79,E2 -14877.79} C_VEL
LIN {X 0,Y 343.38,Z 663.696,A -85,B 0,C 180,E1 -14878.663,E2 -14878.663} C_VEL
LIN {X 0,Y 344.602,Z 648.665,A -85,B 0,C 180,E1 -14879.303,E2 -14879.303} C_VEL
LIN {X 0,Y 345.411,Z 633.024,A -85,B 0,C 180,E1 -14879.73,E2 -14879.73} C_VEL
LIN {X 0,Y 348.759,Z 521.25,A -85,B 0,C 180,E1 -14882.033,E2 -14882.033} C_VEL
LIN {X 0,Y 349.003,Z 506.976,A -85,B 0,C 180,E1 -14882.347,E2 -14882.347} C_VEL
LIN {X 0,Y 345.263,Z 476.017,A -85,B 0,C 180,E1 -14883.495,E2 -14883.495} C_VEL
LIN {X 0,Y 343.994,Z 465.837,A -85,B 0,C 180,E1 -14883.925,E2 -14883.925} C_VEL
LIN {X 0,Y 342.896,Z 439.766,A -85,B 0,C 180,E1 -14885.755,E2 -14885.755} C_VEL
LIN {X 0,Y 336.569,Z 422.42,A -85,B 0,C 180,E1 -14887.706,E2 -14887.706} C_VEL
LIN {X 0,Y 333.262,Z 413.524,A -85,B 0,C 180,E1 -14888.82,E2 -14888.82} C_VEL
LIN {X 0,Y 328.349,Z 396.741,A -85,B 0,C 180,E1 -14892.088,E2 -14892.088} C_VEL
LIN {X 0,Y 326.61,Z 390.579,A -85,B 0,C 180,E1 -14893.396,E2 -14893.396} C_VEL
LIN {X 0,Y 326.56,Z 390.388,A -85,B 0,C 180,E1 -14897.028,E2 -14897.028} C_VEL
LIN {X 0,Y 326.569,Z 390.432,A -85,B 0,C 180,E1 -14901.384,E2 -14901.384} C_VEL
LIN {X 0,Y 326.604,Z 390.369,A -85,B 0,C 180,E1 -14904.851,E2 -14904.851} C_VEL
LIN {X 0,Y 326.595,Z 390.412,A -85,B 0,C 180,E1 -14907.454,E2 -14907.454} C_VEL
LIN {X 0,Y 326.568,Z 390.417,A -85,B 0,C 180,E1 -14910.332,E2 -14910.332} C_VEL
LIN {X 0,Y 326.588,Z 390.429,A -85,B 0,C 180,E1 -14913.134,E2 -14913.134} C_VEL
LIN {X 0,Y 326.577,Z 390.43,A -85,B 0,C 180,E1 -14917.21,E2 -14917.21} C_VEL
LIN {X 0,Y 326.633,Z 390.413,A -85,B 0,C 180,E1 -14921.205,E2 -14921.205} C_VEL
LIN {X 0,Y 326.71,Z 390.393,A -85,B 0,C 180,E1 -14925.459,E2 -14925.459} C_VEL
LIN {X 0,Y 326.741,Z 390.402,A -85,B 0,C 180,E1 -14928.838,E2 -14928.838} C_VEL
LIN {X 0,Y 326.895,Z 390.388,A -85,B 0,C 180,E1 -14932.589,E2 -14932.589} C_VEL
LIN {X 0,Y 326.735,Z 390.391,A -85,B 0,C 180,E1 -14935.064,E2 -14935.064} C_VEL
LIN {X 0,Y 326.997,Z 390.373,A -85,B 0,C 180,E1 -14937.537,E2 -14937.537} C_VEL
LIN {X 0,Y 327.032,Z 390.351,A -85,B 0,C 180,E1 -14941.232,E2 -14941.232} C_VEL
LIN {X 0,Y 326.74,Z 390.409,A -85,B 0,C 180,E1 -14943.7,E2 -14943.7} C_VEL
LIN {X 0,Y 326.907,Z 390.368,A -85,B 0,C 180,E1 -14946.705,E2 -14946.705} C_VEL
LIN {X 0,Y 326.768,Z 390.404,A -85,B 0,C 180,E1 -14949.908,E2 -14949.908} C_VEL
LIN {X 0,Y 326.744,Z 390.405,A -85,B 0,C 180,E1 -14953.686,E2 -14953.686} C_VEL
LIN {X 0,Y 326.649,Z 390.407,A -85,B 0,C 180,E1 -14957.531,E2 -14957.531} C_VEL
LIN {X 0,Y 326.6,Z 390.411,A -85,B 0,C 180,E1 -14961.458,E2 -14961.458} C_VEL
LIN {X 0,Y 326.587,Z 390.414,A -85,B 0,C 180,E1 -14965.493,E2 -14965.493} C_VEL
LIN {X 0,Y 326.576,Z 390.425,A -85,B 0,C 180,E1 -14968.258,E2 -14968.258} C_VEL
LIN {X 0,Y 326.555,Z 390.437,A -85,B 0,C 180,E1 -14971.099,E2 -14971.099} C_VEL
LIN {X 0,Y 326.593,Z 390.43,A -85,B 0,C 180,E1 -14974.021,E2 -14974.021} C_VEL
LIN {X 0,Y 326.61,Z 390.387,A -85,B 0,C 180,E1 -14977.239,E2 -14977.239} C_VEL
LIN {X 0,Y 326.602,Z 390.612,A -85,B 0,C 180,E1 -14981.023,E2 -14981.023} C_VEL
LIN {X 0,Y 327.529,Z 393.129,A -85,B 0,C 180,E1 -14981.697,E2 -14981.697} C_VEL
LIN {X 0,Y 332.746,Z 405.474,A -85,B 0,C 180,E1 -14984.61,E2 -14984.61} C_VEL
LIN {X 0,Y 336.724,Z 416.154,A -85,B 0,C 180,E1 -14986.929,E2 -14986.929} C_VEL
LIN {X 0,Y 341.132,Z 429.71,A -85,B 0,C 180,E1 -14989.665,E2 -14989.665} C_VEL
LIN {X 0,Y 345.207,Z 444.198,A -85,B 0,C 180,E1 -14992.358,E2 -14992.358} C_VEL
LIN {X 0,Y 345.776,Z 447.247,A -85,B 0,C 180,E1 -14992.875,E2 -14992.875} C_VEL
LIN {X 0,Y 343.753,Z 468.344,A -85,B 0,C 180,E1 -14995.615,E2 -14995.615} C_VEL
LIN {X 0,Y 343.548,Z 471.432,A -85,B 0,C 180,E1 -14995.967,E2 -14995.967} C_VEL
LIN {X 0,Y 348.354,Z 502.093,A -85,B 0,C 180,E1 -14997.244,E2 -14997.244} C_VEL
LIN {X 0,Y 349.72,Z 512.494,A -85,B 0,C 180,E1 -14997.635,E2 -14997.635} C_VEL
LIN {X 0,Y 345.658,Z 640.266,A -85,B 0,C 180,E1 -15000.293,E2 -15000.293} C_VEL
LIN {X 0,Y 344.659,Z 655.873,A -85,B 0,C 180,E1 -15000.828,E2 -15000.828} C_VEL
LIN {X 0,Y 343.324,Z 669.586,A -85,B 0,C 180,E1 -15001.499,E2 -15001.499} C_VEL
LIN {X 0,Y 341.605,Z 684.202,A -85,B 0,C 180,E1 -15002.458,E2 -15002.458} C_VEL
LIN {X 0,Y 339.755,Z 697.703,A -85,B 0,C 180,E1 -15003.596,E2 -15003.596} C_VEL
LIN {X 0,Y 337.403,Z 711.669,A -85,B 0,C 180,E1 -15005.054,E2 -15005.054} C_VEL
LIN {X 0,Y 335.192,Z 724.26,A -85,B 0,C 180,E1 -15006.689,E2 -15006.689} C_VEL
LIN {X 0,Y 333.095,Z 735.828,A -85,B 0,C 180,E1 -15008.522,E2 -15008.522} C_VEL
LIN {X 0,Y 330.954,Z 746.05,A -85,B 0,C 180,E1 -15010.463,E2 -15010.463} C_VEL
LIN {X 0,Y 329.18,Z 755.358,A -85,B 0,C 180,E1 -15012.611,E2 -15012.611} C_VEL
LIN {X 0,Y 327.736,Z 763.167,A -85,B 0,C 180,E1 -15014.793,E2 -15014.793} C_VEL
LIN {X 0,Y 326.675,Z 769.528,A -85,B 0,C 180,E1 -15016.947,E2 -15016.947} C_VEL
LIN {X 0,Y 325.724,Z 775.422,A -85,B 0,C 180,E1 -15019.434,E2 -15019.434} C_VEL
LIN {X 0,Y 325.307,Z 778.899,A -85,B 0,C 180,E1 -15021.304,E2 -15021.304} C_VEL
LIN {X 0,Y 324.953,Z 782.442,A -85,B 0,C 180,E1 -15023.794,E2 -15023.794} C_VEL
LIN {X 0,Y 324.846,Z 784.783,A -85,B 0,C 180,E1 -15026.281,E2 -15026.281} C_VEL
LIN {X 0,Y 324.773,Z 785.975,A -85,B 0,C 180,E1 -15028.762,E2 -15028.762} C_VEL
LIN {X 0,Y 324.774,Z 785.989,A -85,B 0,C 180,E1 -15031.242,E2 -15031.242} C_VEL
LIN {X 0,Y 324.85,Z 784.852,A -85,B 0,C 180,E1 -15033.723,E2 -15033.723} C_VEL
LIN {X 0,Y 324.96,Z 782.563,A -85,B 0,C 180,E1 -15036.21,E2 -15036.21} C_VEL
LIN {X 0,Y 325.31,Z 779.068,A -85,B 0,C 180,E1 -15038.7,E2 -15038.7} C_VEL
LIN {X 0,Y 325.86,Z 774.288,A -85,B 0,C 180,E1 -15041.194,E2 -15041.194} C_VEL
LIN {X 0,Y 326.904,Z 768.101,A -85,B 0,C 180,E1 -15043.681,E2 -15043.681} C_VEL
LIN {X 0,Y 328.257,Z 760.317,A -85,B 0,C 180,E1 -15046.162,E2 -15046.162} C_VEL
LIN {X 0,Y 329.844,Z 752.014,A -85,B 0,C 180,E1 -15048.319,E2 -15048.319} C_VEL
LIN {X 0,Y 331.553,Z 743.587,A -85,B 0,C 180,E1 -15050.15,E2 -15050.15} C_VEL
LIN {X 0,Y 333.815,Z 731.798,A -85,B 0,C 180,E1 -15052.271,E2 -15052.271} C_VEL
LIN {X 0,Y 336.086,Z 719.559,A -85,B 0,C 180,E1 -15054.067,E2 -15054.067} C_VEL
LIN {X 0,Y 338.21,Z 707.323,A -85,B 0,C 180,E1 -15055.544,E2 -15055.544} C_VEL
LIN {X 0,Y 340.368,Z 693.964,A -85,B 0,C 180,E1 -15056.853,E2 -15056.853} C_VEL
LIN {X 0,Y 342.212,Z 680.061,A -85,B 0,C 180,E1 -15057.947,E2 -15057.947} C_VEL
LIN {X 0,Y 342.814,Z 674.773,A -85,B 0,C 180,E1 -15058.297,E2 -15058.297} C_VEL
LIN {X 0,Y 342.852,Z 669.332,A -85,B 0,C 180,E1 -15058.684,E2 -15058.684} C_VEL
LIN {X 0,Y 341.206,Z 660.454,A -85,B 0,C 180,E1 -15059.373,E2 -15059.373} C_VEL
LIN {X 0,Y 339.482,Z 651.411,A -85,B 0,C 180,E1 -15059.988,E2 -15059.988} C_VEL
LIN {X 0,Y 339.285,Z 645.715,A -85,B 0,C 180,E1 -15060.24,E2 -15060.24} C_VEL
LIN {X 0,Y 340.015,Z 628.203,A -85,B 0,C 180,E1 -15060.684,E2 -15060.684} C_VEL
LIN {X 0,Y 343.141,Z 531.652,A -85,B 0,C 180,E1 -15062.704,E2 -15062.704} C_VEL
LIN {X 0,Y 343.644,Z 512.024,A -85,B 0,C 180,E1 -15063.129,E2 -15063.129} C_VEL
LIN {X 0,Y 339.115,Z 481.285,A -85,B 0,C 180,E1 -15064.397,E2 -15064.397} C_VEL
LIN {X 0,Y 337.51,Z 470.948,A -85,B 0,C 180,E1 -15064.87,E2 -15064.87} C_VEL
LIN {X 0,Y 339.509,Z 450.794,A -85,B 0,C 180,E1 -15067.485,E2 -15067.485} C_VEL
LIN {X 0,Y 339.071,Z 447.435,A -85,B 0,C 180,E1 -15068.035,E2 -15068.035} C_VEL
LIN {X 0,Y 334.93,Z 432.135,A -85,B 0,C 180,E1 -15070.939,E2 -15070.939} C_VEL
LIN {X 0,Y 330.534,Z 418.725,A -85,B 0,C 180,E1 -15073.703,E2 -15073.703} C_VEL
LIN {X 0,Y 324.887,Z 404.032,A -85,B 0,C 180,E1 -15077.047,E2 -15077.047} C_VEL
LIN {X 0,Y 320.896,Z 394.707,A -85,B 0,C 180,E1 -15079.341,E2 -15079.341} C_VEL
LIN {X 0,Y 319.536,Z 391.486,A -85,B 0,C 180,E1 -15080.245,E2 -15080.245} C_VEL
LIN {X 0,Y 319.56,Z 391.282,A -85,B 0,C 180,E1 -15083.572,E2 -15083.572} C_VEL
LIN {X 0,Y 319.583,Z 391.275,A -85,B 0,C 180,E1 -15086.687,E2 -15086.687} C_VEL
LIN {X 0,Y 319.598,Z 391.485,A -85,B 0,C 180,E1 -15090.797,E2 -15090.797} C_VEL
LIN {X 0,Y 320.312,Z 394.358,A -85,B 0,C 180,E1 -15091.466,E2 -15091.466} C_VEL
LIN {X 0,Y 332.512,Z 426.332,A -85,B 0,C 180,E1 -15093.344,E2 -15093.344} C_VEL
LIN {X 0,Y 328.225,Z 537.855,A -85,B 0,C 180,E1 -15096.706,E2 -15096.706} C_VEL
LIN {X 0,Y 327.723,Z 553.102,A -85,B 0,C 180,E1 -15097.397,E2 -15097.397} C_VEL
LIN {X 0,Y 326.983,Z 568.066,A -85,B 0,C 180,E1 -15098.32,E2 -15098.32} C_VEL
LIN {X 0,Y 326.099,Z 581.012,A -85,B 0,C 180,E1 -15099.334,E2 -15099.334} C_VEL
LIN {X 0,Y 325.243,Z 594.008,A -85,B 0,C 180,E1 -15100.596,E2 -15100.596} C_VEL
LIN {X 0,Y 324.134,Z 607.309,A -85,B 0,C 180,E1 -15102.166,E2 -15102.166} C_VEL
LIN {X 0,Y 323.211,Z 619.3,A -85,B 0,C 180,E1 -15103.904,E2 -15103.904} C_VEL
LIN {X 0,Y 322.166,Z 630.123,A -85,B 0,C 180,E1 -15105.793,E2 -15105.793} C_VEL
LIN {X 0,Y 321.476,Z 639.166,A -85,B 0,C 180,E1 -15107.693,E2 -15107.693} C_VEL
LIN {X 0,Y 320.794,Z 647.908,A -85,B 0,C 180,E1 -15109.906,E2 -15109.906} C_VEL
LIN {X 0,Y 320.407,Z 654.038,A -85,B 0,C 180,E1 -15111.803,E2 -15111.803} C_VEL
LIN {X 0,Y 320.063,Z 659.125,A -85,B 0,C 180,E1 -15113.697,E2 -15113.697} C_VEL
LIN {X 0,Y 319.796,Z 663.29,A -85,B 0,C 180,E1 -15115.588,E2 -15115.588} C_VEL
LIN {X 0,Y 319.868,Z 666.497,A -85,B 0,C 180,E1 -15117.481,E2 -15117.481} C_VEL
LIN {X 0,Y 319.928,Z 668.185,A -85,B 0,C 180,E1 -15118.741,E2 -15118.741} C_VEL
LIN {X 0,Y 319.939,Z 669.517,A -85,B 0,C 180,E1 -15120,E2 -15120} C_VEL
LIN {X 0,Y 320.279,Z 670.446,A -85,B 0,C 180,E1 -15121.257,E2 -15121.257} C_VEL
LIN {X 0,Y 320.906,Z 671.257,A -85,B 0,C 180,E1 -15123.767,E2 -15123.767} C_VEL
LIN {X 0,Y 321.664,Z 670.667,A -85,B 0,C 180,E1 -15126.272,E2 -15126.272} C_VEL
LIN {X 0,Y 322.888,Z 668.636,A -85,B 0,C 180,E1 -15128.764,E2 -15128.764} C_VEL
LIN {X 0,Y 324.389,Z 665.164,A -85,B 0,C 180,E1 -15131.244,E2 -15131.244} C_VEL
LIN {X 0,Y 326.379,Z 660.066,A -85,B 0,C 180,E1 -15133.702,E2 -15133.702} C_VEL
LIN {X 0,Y 328.342,Z 654.333,A -85,B 0,C 180,E1 -15135.805,E2 -15135.805} C_VEL
LIN {X 0,Y 330.625,Z 646.885,A -85,B 0,C 180,E1 -15137.952,E2 -15137.952} C_VEL
LIN {X 0,Y 333.177,Z 637.818,A -85,B 0,C 180,E1 -15140.046,E2 -15140.046} C_VEL
LIN {X 0,Y 335.678,Z 628.361,A -85,B 0,C 180,E1 -15141.816,E2 -15141.816} C_VEL
LIN {X 0,Y 338.551,Z 616.021,A -85,B 0,C 180,E1 -15143.716,E2 -15143.716} C_VEL
LIN {X 0,Y 341.154,Z 603.175,A -85,B 0,C 180,E1 -15145.306,E2 -15145.306} C_VEL
LIN {X 0,Y 343.772,Z 588.854,A -85,B 0,C 180,E1 -15146.728,E2 -15146.728} C_VEL
LIN {X 0,Y 345.994,Z 573.524,A -85,B 0,C 180,E1 -15147.934,E2 -15147.934} C_VEL
LIN {X 0,Y 347.953,Z 556.925,A -85,B 0,C 180,E1 -15148.914,E2 -15148.914} C_VEL
LIN {X 0,Y 349.76,Z 539.104,A -85,B 0,C 180,E1 -15149.724,E2 -15149.724} C_VEL
LIN {X 0,Y 355.852,Z 494.583,A -85,B 0,C 180,E1 -15151.491,E2 -15151.491} C_VEL
LIN {X 0,Y 361.317,Z 458.591,A -85,B 0,C 180,E1 -15152.896,E2 -15152.896} C_VEL
LIN {X 0,Y 358.359,Z 453.786,A -85,B 0,C 180,E1 -15154.31,E2 -15154.31} C_VEL
LIN {X 0,Y 356.425,Z 451.035,A -85,B 0,C 180,E1 -15155.363,E2 -15155.363} C_VEL
LIN {X 0,Y 354.634,Z 448.715,A -85,B 0,C 180,E1 -15156.479,E2 -15156.479} C_VEL
LIN {X 0,Y 352.734,Z 446.415,A -85,B 0,C 180,E1 -15157.949,E2 -15157.949} C_VEL
LIN {X 0,Y 350.609,Z 444.602,A -85,B 0,C 180,E1 -15160.383,E2 -15160.383} C_VEL
LIN {X 0,Y 349.735,Z 444.998,A -85,B 0,C 180,E1 -15162.568,E2 -15162.568} C_VEL
LIN {X 0,Y 349.939,Z 446.542,A -85,B 0,C 180,E1 -15164.575,E2 -15164.575} C_VEL
LIN {X 0,Y 350.902,Z 449.441,A -85,B 0,C 180,E1 -15166.474,E2 -15166.474} C_VEL
LIN {X 0,Y 352.806,Z 454.011,A -85,B 0,C 180,E1 -15168.486,E2 -15168.486} C_VEL
LIN {X 0,Y 354.924,Z 459.967,A -85,B 0,C 180,E1 -15170.175,E2 -15170.175} C_VEL
LIN {X 0,Y 356.094,Z 463.309,A -85,B 0,C 180,E1 -15170.962,E2 -15170.962} C_VEL
LIN {X 0,Y 356.338,Z 477.64,A -85,B 0,C 180,E1 -15172.307,E2 -15172.307} C_VEL
LIN {X 0,Y 356.365,Z 492.917,A -85,B 0,C 180,E1 -15173.493,E2 -15173.493} C_VEL
LIN {X 0,Y 355.996,Z 506.766,A -85,B 0,C 180,E1 -15174.367,E2 -15174.367} C_VEL
LIN {X 0,Y 355.48,Z 514.476,A -85,B 0,C 180,E1 -15174.756,E2 -15174.756} C_VEL
LIN {X 0,Y 347.776,Z 581.733,A -85,B 0,C 180,E1 -15177.103,E2 -15177.103} C_VEL
LIN {X 0,Y 344.767,Z 609.122,A -85,B 0,C 180,E1 -15178.079,E2 -15178.079} C_VEL
LIN {X 0,Y 342.048,Z 626.752,A -85,B 0,C 180,E1 -15178.918,E2 -15178.918} C_VEL
LIN {X 0,Y 338.818,Z 643.593,A -85,B 0,C 180,E1 -15179.928,E2 -15179.928} C_VEL
LIN {X 0,Y 337.7,Z 658.758,A -85,B 0,C 180,E1 -15180.505,E2 -15180.505} C_VEL
LIN {X 0,Y 336.262,Z 672.916,A -85,B 0,C 180,E1 -15181.267,E2 -15181.267} C_VEL
LIN {X 0,Y 334.523,Z 687.071,A -85,B 0,C 180,E1 -15182.277,E2 -15182.277} C_VEL
LIN {X 0,Y 332.514,Z 700.414,A -85,B 0,C 180,E1 -15183.479,E2 -15183.479} C_VEL
LIN {X 0,Y 330.245,Z 713.742,A -85,B 0,C 180,E1 -15184.976,E2 -15184.976} C_VEL
LIN {X 0,Y 327.9,Z 725.861,A -85,B 0,C 180,E1 -15186.638,E2 -15186.638} C_VEL
LIN {X 0,Y 325.791,Z 736.91,A -85,B 0,C 180,E1 -15188.484,E2 -15188.484} C_VEL
LIN {X 0,Y 323.837,Z 746.203,A -85,B 0,C 180,E1 -15190.341,E2 -15190.341} C_VEL
LIN {X 0,Y 322.057,Z 755.318,A -85,B 0,C 180,E1 -15192.537,E2 -15192.537} C_VEL
LIN {X 0,Y 320.528,Z 762.877,A -85,B 0,C 180,E1 -15194.743,E2 -15194.743} C_VEL
LIN {X 0,Y 319.409,Z 769.918,A -85,B 0,C 180,E1 -15197.287,E2 -15197.287} C_VEL
LIN {X 0,Y 318.548,Z 775.448,A -85,B 0,C 180,E1 -15199.832,E2 -15199.832} C_VEL
LIN {X 0,Y 318.122,Z 779.624,A -85,B 0,C 180,E1 -15202.381,E2 -15202.381} C_VEL
LIN {X 0,Y 317.867,Z 782.548,A -85,B 0,C 180,E1 -15204.924,E2 -15204.924} C_VEL
LIN {X 0,Y 317.797,Z 784.288,A -85,B 0,C 180,E1 -15207.463,E2 -15207.463} C_VEL
LIN {X 0,Y 317.769,Z 784.88,A -85,B 0,C 180,E1 -15209.998,E2 -15209.998} C_VEL
LIN {X 0,Y 317.804,Z 784.281,A -85,B 0,C 180,E1 -15212.533,E2 -15212.533} C_VEL
LIN {X 0,Y 317.857,Z 782.532,A -85,B 0,C 180,E1 -15215.072,E2 -15215.072} C_VEL
LIN {X 0,Y 318.081,Z 779.605,A -85,B 0,C 180,E1 -15217.616,E2 -15217.616} C_VEL
LIN {X 0,Y 318.539,Z 775.427,A -85,B 0,C 180,E1 -15220.164,E2 -15220.164} C_VEL
LIN {X 0,Y 319.399,Z 769.886,A -85,B 0,C 180,E1 -15222.709,E2 -15222.709} C_VEL
LIN {X 0,Y 320.522,Z 762.829,A -85,B 0,C 180,E1 -15225.253,E2 -15225.253} C_VEL
LIN {X 0,Y 322.018,Z 755.263,A -85,B 0,C 180,E1 -15227.461,E2 -15227.461} C_VEL
LIN {X 0,Y 323.8,Z 746.14,A -85,B 0,C 180,E1 -15229.657,E2 -15229.657} C_VEL
LIN {X 0,Y 325.757,Z 736.838,A -85,B 0,C 180,E1 -15231.514,E2 -15231.514} C_VEL
LIN {X 0,Y 327.884,Z 725.78,A -85,B 0,C 180,E1 -15233.359,E2 -15233.359} C_VEL
LIN {X 0,Y 330.179,Z 713.646,A -85,B 0,C 180,E1 -15235.025,E2 -15235.025} C_VEL
LIN {X 0,Y 332.468,Z 700.28,A -85,B 0,C 180,E1 -15236.521,E2 -15236.521} C_VEL
LIN {X 0,Y 334.596,Z 685.973,A -85,B 0,C 180,E1 -15237.799,E2 -15237.799} C_VEL
LIN {X 0,Y 336.355,Z 671.55,A -85,B 0,C 180,E1 -15238.806,E2 -15238.806} C_VEL
LIN {X 0,Y 337.843,Z 656.072,A -85,B 0,C 180,E1 -15239.605,E2 -15239.605} C_VEL
LIN {X 0,Y 338.918,Z 640.639,A -85,B 0,C 180,E1 -15240.144,E2 -15240.144} C_VEL
LIN {X 0,Y 342.434,Z 532.867,A -85,B 0,C 180,E1 -15242.418,E2 -15242.418} C_VEL
LIN {X 0,Y 343.02,Z 508.087,A -85,B 0,C 180,E1 -15242.958,E2 -15242.958} C_VEL
LIN {X 0,Y 339.151,Z 475.53,A -85,B 0,C 180,E1 -15244.196,E2 -15244.196} C_VEL
LIN {X 0,Y 337.963,Z 466.179,A -85,B 0,C 180,E1 -15244.597,E2 -15244.597} C_VEL
LIN {X 0,Y 337.192,Z 442.669,A -85,B 0,C 180,E1 -15246.304,E2 -15246.304} C_VEL
LIN {X 0,Y 331.259,Z 426.072,A -85,B 0,C 180,E1 -15248.219,E2 -15248.219} C_VEL
LIN {X 0,Y 326.353,Z 413.448,A -85,B 0,C 180,E1 -15249.839,E2 -15249.839} C_VEL
LIN {X 0,Y 323.919,Z 406.421,A -85,B 0,C 180,E1 -15250.806,E2 -15250.806} C_VEL
LIN {X 0,Y 319.53,Z 391.507,A -85,B 0,C 180,E1 -15253.902,E2 -15253.902} C_VEL
LIN {X 0,Y 319.538,Z 391.262,A -85,B 0,C 180,E1 -15257.014,E2 -15257.014} C_VEL
LIN {X 0,Y 319.533,Z 391.299,A -85,B 0,C 180,E1 -15260.369,E2 -15260.369} C_VEL
LIN {X 0,Y 319.565,Z 391.244,A -85,B 0,C 180,E1 -15264.456,E2 -15264.456} C_VEL
LIN {X 0,Y 319.511,Z 391.308,A -85,B 0,C 180,E1 -15268.136,E2 -15268.136} C_VEL
LIN {X 0,Y 319.552,Z 391.293,A -85,B 0,C 180,E1 -15271.604,E2 -15271.604} C_VEL
LIN {X 0,Y 319.513,Z 391.291,A -85,B 0,C 180,E1 -15275.297,E2 -15275.297} C_VEL
LIN {X 0,Y 319.548,Z 391.306,A -85,B 0,C 180,E1 -15278.044,E2 -15278.044} C_VEL
LIN {X 0,Y 319.572,Z 391.301,A -85,B 0,C 180,E1 -15282.068,E2 -15282.068} C_VEL
LIN {X 0,Y 319.694,Z 391.271,A -85,B 0,C 180,E1 -15286.006,E2 -15286.006} C_VEL
LIN {X 0,Y 319.719,Z 391.265,A -85,B 0,C 180,E1 -15289.872,E2 -15289.872} C_VEL
LIN {X 0,Y 319.881,Z 391.262,A -85,B 0,C 180,E1 -15293.693,E2 -15293.693} C_VEL
LIN {X 0,Y 319.943,Z 391.25,A -85,B 0,C 180,E1 -15297.482,E2 -15297.482} C_VEL
LIN {X 0,Y 319.999,Z 391.227,A -85,B 0,C 180,E1 -15301.259,E2 -15301.259} C_VEL
LIN {X 0,Y 319.708,Z 391.279,A -85,B 0,C 180,E1 -15305.045,E2 -15305.045} C_VEL
LIN {X 0,Y 319.866,Z 391.25,A -85,B 0,C 180,E1 -15307.576,E2 -15307.576} C_VEL
LIN {X 0,Y 319.699,Z 391.264,A -85,B 0,C 180,E1 -15311.411,E2 -15311.411} C_VEL
LIN {X 0,Y 319.698,Z 391.283,A -85,B 0,C 180,E1 -15314.712,E2 -15314.712} C_VEL
LIN {X 0,Y 319.599,Z 391.29,A -85,B 0,C 180,E1 -15317.93,E2 -15317.93} C_VEL
LIN {X 0,Y 319.551,Z 391.292,A -85,B 0,C 180,E1 -15321.956,E2 -15321.956} C_VEL
LIN {X 0,Y 319.536,Z 391.295,A -85,B 0,C 180,E1 -15326.097,E2 -15326.097} C_VEL
LIN {X 0,Y 319.51,Z 391.3,A -85,B 0,C 180,E1 -15328.942,E2 -15328.942} C_VEL
LIN {X 0,Y 319.507,Z 391.308,A -85,B 0,C 180,E1 -15331.865,E2 -15331.865} C_VEL
LIN {X 0,Y 319.566,Z 391.285,A -85,B 0,C 180,E1 -15335.544,E2 -15335.544} C_VEL
LIN {X 0,Y 319.511,Z 391.272,A -85,B 0,C 180,E1 -15338.017,E2 -15338.017} C_VEL
LIN {X 0,Y 319.522,Z 391.529,A -85,B 0,C 180,E1 -15339.909,E2 -15339.909} C_VEL
LIN {X 0,Y 320.674,Z 394.359,A -85,B 0,C 180,E1 -15340.693,E2 -15340.693} C_VEL
LIN {X 0,Y 325.232,Z 405.008,A -85,B 0,C 180,E1 -15343.321,E2 -15343.321} C_VEL
LIN {X 0,Y 329.78,Z 416.701,A -85,B 0,C 180,E1 -15345.993,E2 -15345.993} C_VEL
LIN {X 0,Y 334.221,Z 430.074,A -85,B 0,C 180,E1 -15348.783,E2 -15348.783} C_VEL
LIN {X 0,Y 338.192,Z 443.894,A -85,B 0,C 180,E1 -15351.436,E2 -15351.436} C_VEL
LIN {X 0,Y 339.487,Z 448.976,A -85,B 0,C 180,E1 -15352.359,E2 -15352.359} C_VEL
LIN {X 0,Y 337.689,Z 468.267,A -85,B 0,C 180,E1 -15354.907,E2 -15354.907} C_VEL
LIN {X 0,Y 337.44,Z 471.44,A -85,B 0,C 180,E1 -15355.268,E2 -15355.268} C_VEL
LIN {X 0,Y 342.329,Z 502.868,A -85,B 0,C 180,E1 -15356.614,E2 -15356.614} C_VEL
LIN {X 0,Y 343.682,Z 513.958,A -85,B 0,C 180,E1 -15357.034,E2 -15357.034} C_VEL
LIN {X 0,Y 339.586,Z 638.814,A -85,B 0,C 180,E1 -15359.664,E2 -15359.664} C_VEL
LIN {X 0,Y 338.647,Z 654.089,A -85,B 0,C 180,E1 -15360.173,E2 -15360.173} C_VEL
LIN {X 0,Y 337.099,Z 669.547,A -85,B 0,C 180,E1 -15360.923,E2 -15360.923} C_VEL
LIN {X 0,Y 335.371,Z 683.768,A -85,B 0,C 180,E1 -15361.866,E2 -15361.866} C_VEL
LIN {X 0,Y 333.371,Z 697.678,A -85,B 0,C 180,E1 -15363.05,E2 -15363.05} C_VEL
LIN {X 0,Y 330.945,Z 711.648,A -85,B 0,C 180,E1 -15364.533,E2 -15364.533} C_VEL
LIN {X 0,Y 328.65,Z 724.241,A -85,B 0,C 180,E1 -15366.197,E2 -15366.197} C_VEL
LIN {X 0,Y 326.699,Z 734.487,A -85,B 0,C 180,E1 -15367.829,E2 -15367.829} C_VEL
LIN {X 0,Y 324.563,Z 744.569,A -85,B 0,C 180,E1 -15369.731,E2 -15369.731} C_VEL
LIN {X 0,Y 322.578,Z 754.128,A -85,B 0,C 180,E1 -15371.915,E2 -15371.915} C_VEL
LIN {X 0,Y 320.952,Z 762.29,A -85,B 0,C 180,E1 -15374.182,E2 -15374.182} C_VEL
LIN {X 0,Y 319.706,Z 769.514,A -85,B 0,C 180,E1 -15376.657,E2 -15376.657} C_VEL
LIN {X 0,Y 318.71,Z 775.408,A -85,B 0,C 180,E1 -15379.199,E2 -15379.199} C_VEL
LIN {X 0,Y 318.273,Z 778.886,A -85,B 0,C 180,E1 -15381.11,E2 -15381.11} C_VEL
LIN {X 0,Y 317.88,Z 782.428,A -85,B 0,C 180,E1 -15383.655,E2 -15383.655} C_VEL
LIN {X 0,Y 317.757,Z 784.77,A -85,B 0,C 180,E1 -15386.198,E2 -15386.198} C_VEL
LIN {X 0,Y 317.687,Z 785.961,A -85,B 0,C 180,E1 -15388.734,E2 -15388.734} C_VEL
LIN {X 0,Y 317.688,Z 785.975,A -85,B 0,C 180,E1 -15391.27,E2 -15391.27} C_VEL
LIN {X 0,Y 317.761,Z 784.837,A -85,B 0,C 180,E1 -15393.806,E2 -15393.806} C_VEL
LIN {X 0,Y 317.887,Z 782.548,A -85,B 0,C 180,E1 -15396.348,E2 -15396.348} C_VEL
LIN {X 0,Y 318.273,Z 779.053,A -85,B 0,C 180,E1 -15398.894,E2 -15398.894} C_VEL
LIN {X 0,Y 318.847,Z 774.272,A -85,B 0,C 180,E1 -15401.444,E2 -15401.444} C_VEL
LIN {X 0,Y 319.94,Z 768.083,A -85,B 0,C 180,E1 -15403.985,E2 -15403.985} C_VEL
LIN {X 0,Y 321.358,Z 760.299,A -85,B 0,C 180,E1 -15406.519,E2 -15406.519} C_VEL
LIN {X 0,Y 323.055,Z 751.994,A -85,B 0,C 180,E1 -15408.718,E2 -15408.718} C_VEL
LIN {X 0,Y 324.864,Z 743.565,A -85,B 0,C 180,E1 -15410.584,E2 -15410.584} C_VEL
LIN {X 0,Y 326.962,Z 733.016,A -85,B 0,C 180,E1 -15412.539,E2 -15412.539} C_VEL
LIN {X 0,Y 329.37,Z 720.676,A -85,B 0,C 180,E1 -15414.421,E2 -15414.421} C_VEL
LIN {X 0,Y 331.791,Z 707.29,A -85,B 0,C 180,E1 -15416.075,E2 -15416.075} C_VEL
LIN {X 0,Y 334.046,Z 693.926,A -85,B 0,C 180,E1 -15417.404,E2 -15417.404} C_VEL
LIN {X 0,Y 335.974,Z 679.801,A -85,B 0,C 180,E1 -15418.53,E2 -15418.53} C_VEL
LIN {X 0,Y 337.527,Z 666.057,A -85,B 0,C 180,E1 -15419.383,E2 -15419.383} C_VEL
LIN {X 0,Y 338.906,Z 650.985,A -85,B 0,C 180,E1 -15420.064,E2 -15420.064} C_VEL
LIN {X 0,Y 339.285,Z 645.715,A -85,B 0,C 180,E1 -15420.24,E2 -15420.24} C_VEL
LIN {X 0,Y 339.065,Z 639.976,A -85,B 0,C 180,E1 -15420.471,E2 -15420.471} C_VEL
LIN {X 0,Y 334.814,Z 621.368,A -85,B 0,C 180,E1 -15421.385,E2 -15421.385} C_VEL
LIN {X 0,Y 334.434,Z 615.564,A -85,B 0,C 180,E1 -15421.562,E2 -15421.562} C_VEL
LIN {X 0,Y 337.796,Z 513.808,A -85,B 0,C 180,E1 -15423.73,E2 -15423.73} C_VEL
LIN {X 0,Y 333.511,Z 484.15,A -85,B 0,C 180,E1 -15424.981,E2 -15424.981} C_VEL
LIN {X 0,Y 331.46,Z 470.769,A -85,B 0,C 180,E1 -15425.61,E2 -15425.61} C_VEL
LIN {X 0,Y 333.33,Z 452.726,A -85,B 0,C 180,E1 -15427.978,E2 -15427.978} C_VEL
LIN {X 0,Y 331.339,Z 444.292,A -85,B 0,C 180,E1 -15429.52,E2 -15429.52} C_VEL
LIN {X 0,Y 327.928,Z 432.237,A -85,B 0,C 180,E1 -15431.911,E2 -15431.911} C_VEL
LIN {X 0,Y 324.159,Z 420.973,A -85,B 0,C 180,E1 -15434.319,E2 -15434.319} C_VEL
LIN {X 0,Y 319.335,Z 408.254,A -85,B 0,C 180,E1 -15437.274,E2 -15437.274} C_VEL
LIN {X 0,Y 314.307,Z 396.766,A -85,B 0,C 180,E1 -15440.202,E2 -15440.202} C_VEL
LIN {X 0,Y 312.514,Z 392.536,A -85,B 0,C 180,E1 -15441.374,E2 -15441.374} C_VEL
LIN {X 0,Y 312.481,Z 392.176,A -85,B 0,C 180,E1 -15441.925,E2 -15441.925} C_VEL
LIN {X 0,Y 312.535,Z 392.145,A -85,B 0,C 180,E1 -15444.221,E2 -15444.221} C_VEL
LIN {X 0,Y 312.505,Z 392.168,A -85,B 0,C 180,E1 -15447.334,E2 -15447.334} C_VEL
LIN {X 0,Y 312.571,Z 392.351,A -85,B 0,C 180,E1 -15450.378,E2 -15450.378} C_VEL
LIN {X 0,Y 313.167,Z 394.834,A -85,B 0,C 180,E1 -15450.986,E2 -15450.986} C_VEL
LIN {X 0,Y 325.814,Z 428.171,A -85,B 0,C 180,E1 -15452.991,E2 -15452.991} C_VEL
LIN {X 0,Y 321.36,Z 538.087,A -85,B 0,C 180,E1 -15456.391,E2 -15456.391} C_VEL
LIN {X 0,Y 320.849,Z 553.058,A -85,B 0,C 180,E1 -15457.072,E2 -15457.072} C_VEL
LIN {X 0,Y 320.123,Z 568.023,A -85,B 0,C 180,E1 -15458.007,E2 -15458.007} C_VEL
LIN {X 0,Y 319.126,Z 582.835,A -85,B 0,C 180,E1 -15459.199,E2 -15459.199} C_VEL
LIN {X 0,Y 318.122,Z 597.095,A -85,B 0,C 180,E1 -15460.647,E2 -15460.647} C_VEL
LIN {X 0,Y 316.978,Z 609.929,A -85,B 0,C 180,E1 -15462.253,E2 -15462.253} C_VEL
LIN {X 0,Y 316.126,Z 620.662,A -85,B 0,C 180,E1 -15463.865,E2 -15463.865} C_VEL
LIN {X 0,Y 315.082,Z 631.456,A -85,B 0,C 180,E1 -15465.797,E2 -15465.797} C_VEL
LIN {X 0,Y 314.406,Z 640.489,A -85,B 0,C 180,E1 -15467.739,E2 -15467.739} C_VEL
LIN {X 0,Y 313.804,Z 648.058,A -85,B 0,C 180,E1 -15469.678,E2 -15469.678} C_VEL
LIN {X 0,Y 313.365,Z 654.39,A -85,B 0,C 180,E1 -15471.617,E2 -15471.617} C_VEL
LIN {X 0,Y 313.035,Z 659.655,A -85,B 0,C 180,E1 -15473.555,E2 -15473.555} C_VEL
LIN {X 0,Y 312.763,Z 663.945,A -85,B 0,C 180,E1 -15475.489,E2 -15475.489} C_VEL
LIN {X 0,Y 312.814,Z 667.259,A -85,B 0,C 180,E1 -15477.424,E2 -15477.424} C_VEL
LIN {X 0,Y 312.902,Z 669.022,A -85,B 0,C 180,E1 -15478.713,E2 -15478.713} C_VEL
LIN {X 0,Y 312.91,Z 670.445,A -85,B 0,C 180,E1 -15480,E2 -15480} C_VEL
LIN {X 0,Y 313.278,Z 671.471,A -85,B 0,C 180,E1 -15481.285,E2 -15481.285} C_VEL
LIN {X 0,Y 313.942,Z 672.482,A -85,B 0,C 180,E1 -15483.851,E2 -15483.851} C_VEL
LIN {X 0,Y 314.747,Z 672.081,A -85,B 0,C 180,E1 -15486.41,E2 -15486.41} C_VEL
LIN {X 0,Y 316.065,Z 670.221,A -85,B 0,C 180,E1 -15488.954,E2 -15488.954} C_VEL
LIN {X 0,Y 317.642,Z 666.907,A -85,B 0,C 180,E1 -15491.486,E2 -15491.486} C_VEL
LIN {X 0,Y 319.76,Z 662.059,A -85,B 0,C 180,E1 -15493.991,E2 -15493.991} C_VEL
LIN {X 0,Y 321.692,Z 656.898,A -85,B 0,C 180,E1 -15495.995,E2 -15495.995} C_VEL
LIN {X 0,Y 324.267,Z 649.373,A -85,B 0,C 180,E1 -15498.316,E2 -15498.316} C_VEL
LIN {X 0,Y 326.988,Z 640.629,A -85,B 0,C 180,E1 -15500.442,E2 -15500.442} C_VEL
LIN {X 0,Y 330.076,Z 629.852,A -85,B 0,C 180,E1 -15502.535,E2 -15502.535} C_VEL
LIN {X 0,Y 332.991,Z 618.367,A -85,B 0,C 180,E1 -15504.352,E2 -15504.352} C_VEL
LIN {X 0,Y 335.96,Z 605.033,A -85,B 0,C 180,E1 -15506.059,E2 -15506.059} C_VEL
LIN {X 0,Y 338.443,Z 592.493,A -85,B 0,C 180,E1 -15507.351,E2 -15507.351} C_VEL
LIN {X 0,Y 340.998,Z 577.055,A -85,B 0,C 180,E1 -15508.632,E2 -15508.632} C_VEL
LIN {X 0,Y 343.16,Z 561.047,A -85,B 0,C 180,E1 -15509.652,E2 -15509.652} C_VEL
LIN {X 0,Y 345.204,Z 542.394,A -85,B 0,C 180,E1 -15510.553,E2 -15510.553} C_VEL
LIN {X 0,Y 351.949,Z 496.603,A -85,B 0,C 180,E1 -15512.414,E2 -15512.414} C_VEL
LIN {X 0,Y 357.415,Z 462.838,A -85,B 0,C 180,E1 -15513.75,E2 -15513.75} C_VEL
LIN {X 0,Y 354.647,Z 458.269,A -85,B 0,C 180,E1 -15515.275,E2 -15515.275} C_VEL
LIN {X 0,Y 352.345,Z 455.238,A -85,B 0,C 180,E1 -15516.755,E2 -15516.755} C_VEL
LIN {X 0,Y 350.712,Z 453.148,A -85,B 0,C 180,E1 -15518.104,E2 -15518.104} C_VEL
LIN {X 0,Y 348.962,Z 451.538,A -85,B 0,C 180,E1 -15520.126,E2 -15520.126} C_VEL
LIN {X 0,Y 347.999,Z 451.754,A -85,B 0,C 180,E1 -15522.26,E2 -15522.26} C_VEL
LIN {X 0,Y 348.017,Z 453.12,A -85,B 0,C 180,E1 -15524.193,E2 -15524.193} C_VEL
LIN {X 0,Y 348.725,Z 455.55,A -85,B 0,C 180,E1 -15525.932,E2 -15525.932} C_VEL
LIN {X 0,Y 350.247,Z 459.695,A -85,B 0,C 180,E1 -15527.868,E2 -15527.868} C_VEL
LIN {X 0,Y 351.487,Z 463.531,A -85,B 0,C 180,E1 -15529.078,E2 -15529.078} C_VEL
LIN {X 0,Y 352.958,Z 468.188,A -85,B 0,C 180,E1 -15530.257,E2 -15530.257} C_VEL
LIN {X 0,Y 352.789,Z 484.364,A -85,B 0,C 180,E1 -15531.754,E2 -15531.754} C_VEL
LIN {X 0,Y 352.45,Z 497.867,A -85,B 0,C 180,E1 -15532.781,E2 -15532.781} C_VEL
LIN {X 0,Y 351.78,Z 512.024,A -85,B 0,C 180,E1 -15533.667,E2 -15533.667} C_VEL
LIN {X 0,Y 350.161,Z 524.798,A -85,B 0,C 180,E1 -15534.162,E2 -15534.162} C_VEL
LIN {X 0,Y 342.125,Z 591.174,A -85,B 0,C 180,E1 -15536.533,E2 -15536.533} C_VEL
LIN {X 0,Y 339.689,Z 610.602,A -85,B 0,C 180,E1 -15537.28,E2 -15537.28} C_VEL
LIN {X 0,Y 336.596,Z 628.22,A -85,B 0,C 180,E1 -15538.181,E2 -15538.181} C_VEL
LIN {X 0,Y 333.078,Z 644.195,A -85,B 0,C 180,E1 -15539.223,E2 -15539.223} C_VEL
LIN {X 0,Y 332.426,Z 648.116,A -85,B 0,C 180,E1 -15539.464,E2 -15539.464} C_VEL
LIN {X 0,Y 331.088,Z 663.317,A -85,B 0,C 180,E1 -15540.119,E2 -15540.119} C_VEL
LIN {X 0,Y 329.458,Z 677.847,A -85,B 0,C 180,E1 -15540.999,E2 -15540.999} C_VEL
LIN {X 0,Y 327.441,Z 692.584,A -85,B 0,C 180,E1 -15542.17,E2 -15542.17} C_VEL
LIN {X 0,Y 325.179,Z 706.1,A -85,B 0,C 180,E1 -15543.526,E2 -15543.526} C_VEL
LIN {X 0,Y 322.65,Z 719.567,A -85,B 0,C 180,E1 -15545.207,E2 -15545.207} C_VEL
LIN {X 0,Y 320.304,Z 731.082,A -85,B 0,C 180,E1 -15546.969,E2 -15546.969} C_VEL
LIN {X 0,Y 318.168,Z 741.78,A -85,B 0,C 180,E1 -15548.963,E2 -15548.963} C_VEL
LIN {X 0,Y 316.004,Z 751.657,A -85,B 0,C 180,E1 -15551.185,E2 -15551.185} C_VEL
LIN {X 0,Y 314.283,Z 759.849,A -85,B 0,C 180,E1 -15553.432,E2 -15553.432} C_VEL
LIN {X 0,Y 312.961,Z 766.616,A -85,B 0,C 180,E1 -15555.697,E2 -15555.697} C_VEL
LIN {X 0,Y 311.868,Z 772.876,A -85,B 0,C 180,E1 -15558.296,E2 -15558.296} C_VEL
LIN {X 0,Y 311.247,Z 777.713,A -85,B 0,C 180,E1 -15560.904,E2 -15560.904} C_VEL
LIN {X 0,Y 310.9,Z 781.252,A -85,B 0,C 180,E1 -15563.508,E2 -15563.508} C_VEL
LIN {X 0,Y 310.758,Z 783.577,A -85,B 0,C 180,E1 -15566.108,E2 -15566.108} C_VEL
LIN {X 0,Y 310.672,Z 784.742,A -85,B 0,C 180,E1 -15568.702,E2 -15568.702} C_VEL
LIN {X 0,Y 310.675,Z 784.74,A -85,B 0,C 180,E1 -15571.294,E2 -15571.294} C_VEL
LIN {X 0,Y 310.756,Z 783.564,A -85,B 0,C 180,E1 -15573.888,E2 -15573.888} C_VEL
LIN {X 0,Y 310.892,Z 781.233,A -85,B 0,C 180,E1 -15576.488,E2 -15576.488} C_VEL
LIN {X 0,Y 311.241,Z 777.692,A -85,B 0,C 180,E1 -15579.092,E2 -15579.092} C_VEL
LIN {X 0,Y 311.86,Z 772.849,A -85,B 0,C 180,E1 -15581.7,E2 -15581.7} C_VEL
LIN {X 0,Y 312.947,Z 766.573,A -85,B 0,C 180,E1 -15584.3,E2 -15584.3} C_VEL
LIN {X 0,Y 314.479,Z 758.683,A -85,B 0,C 180,E1 -15586.887,E2 -15586.887} C_VEL
LIN {X 0,Y 316.244,Z 750.259,A -85,B 0,C 180,E1 -15589.133,E2 -15589.133} C_VEL
LIN {X 0,Y 318.145,Z 741.708,A -85,B 0,C 180,E1 -15591.035,E2 -15591.035} C_VEL
LIN {X 0,Y 320.263,Z 731.104,A -85,B 0,C 180,E1 -15593.01,E2 -15593.01} C_VEL
LIN {X 0,Y 322.583,Z 719.473,A -85,B 0,C 180,E1 -15594.794,E2 -15594.794} C_VEL
LIN {X 0,Y 324.895,Z 707.315,A -85,B 0,C 180,E1 -15596.322,E2 -15596.322} C_VEL
LIN {X 0,Y 327.081,Z 694.061,A -85,B 0,C 180,E1 -15597.685,E2 -15597.685} C_VEL
LIN {X 0,Y 329.224,Z 679.232,A -85,B 0,C 180,E1 -15598.892,E2 -15598.892} C_VEL
LIN {X 0,Y 330.837,Z 665.183,A -85,B 0,C 180,E1 -15599.77,E2 -15599.77} C_VEL
LIN {X 0,Y 332.229,Z 649.834,A -85,B 0,C 180,E1 -15600.464,E2 -15600.464} C_VEL
LIN {X 0,Y 333.117,Z 634.901,A -85,B 0,C 180,E1 -15600.901,E2 -15600.901} C_VEL
LIN {X 0,Y 336.719,Z 525.063,A -85,B 0,C 180,E1 -15603.235,E2 -15603.235} C_VEL
LIN {X 0,Y 337.049,Z 508.751,A -85,B 0,C 180,E1 -15603.605,E2 -15603.605} C_VEL
LIN {X 0,Y 333.382,Z 477.359,A -85,B 0,C 180,E1 -15604.829,E2 -15604.829} C_VEL
LIN {X 0,Y 332.018,Z 466.888,A -85,B 0,C 180,E1 -15605.266,E2 -15605.266} C_VEL
LIN {X 0,Y 331.522,Z 446.068,A -85,B 0,C 180,E1 -15606.82,E2 -15606.82} C_VEL
LIN {X 0,Y 328.515,Z 436.987,A -85,B 0,C 180,E1 -15607.857,E2 -15607.857} C_VEL
LIN {X 0,Y 322.493,Z 420.39,A -85,B 0,C 180,E1 -15609.958,E2 -15609.958} C_VEL
LIN {X 0,Y 317.232,Z 406.556,A -85,B 0,C 180,E1 -15611.897,E2 -15611.897} C_VEL
LIN {X 0,Y 314.259,Z 398.271,A -85,B 0,C 180,E1 -15613.146,E2 -15613.146} C_VEL
LIN {X 0,Y 312.481,Z 392.448,A -85,B 0,C 180,E1 -15614.424,E2 -15614.424} C_VEL
LIN {X 0,Y 312.445,Z 392.159,A -85,B 0,C 180,E1 -15616.034,E2 -15616.034} C_VEL
LIN {X 0,Y 312.443,Z 392.166,A -85,B 0,C 180,E1 -15619.884,E2 -15619.884} C_VEL
LIN {X 0,Y 312.52,Z 392.123,A -85,B 0,C 180,E1 -15624.05,E2 -15624.05} C_VEL
LIN {X 0,Y 312.488,Z 392.163,A -85,B 0,C 180,E1 -15627.332,E2 -15627.332} C_VEL
LIN {X 0,Y 312.482,Z 392.171,A -85,B 0,C 180,E1 -15631.294,E2 -15631.294} C_VEL
LIN {X 0,Y 312.503,Z 392.166,A -85,B 0,C 180,E1 -15634.704,E2 -15634.704} C_VEL
LIN {X 0,Y 312.525,Z 392.18,A -85,B 0,C 180,E1 -15637.524,E2 -15637.524} C_VEL
LIN {X 0,Y 312.536,Z 392.174,A -85,B 0,C 180,E1 -15641.65,E2 -15641.65} C_VEL
LIN {X 0,Y 312.636,Z 392.147,A -85,B 0,C 180,E1 -15645.684,E2 -15645.684} C_VEL
LIN {X 0,Y 312.669,Z 392.144,A -85,B 0,C 180,E1 -15649.641,E2 -15649.641} C_VEL
LIN {X 0,Y 312.779,Z 392.142,A -85,B 0,C 180,E1 -15652.252,E2 -15652.252} C_VEL
LIN {X 0,Y 312.674,Z 392.143,A -85,B 0,C 180,E1 -15654.842,E2 -15654.842} C_VEL
LIN {X 0,Y 312.952,Z 392.127,A -85,B 0,C 180,E1 -15658.713,E2 -15658.713} C_VEL
LIN {X 0,Y 312.966,Z 392.102,A -85,B 0,C 180,E1 -15661.287,E2 -15661.287} C_VEL
LIN {X 0,Y 312.837,Z 392.12,A -85,B 0,C 180,E1 -15666.45,E2 -15666.45} C_VEL
LIN {X 0,Y 312.736,Z 392.154,A -85,B 0,C 180,E1 -15669.051,E2 -15669.051} C_VEL
LIN {X 0,Y 312.618,Z 392.154,A -85,B 0,C 180,E1 -15672.992,E2 -15672.992} C_VEL
LIN {X 0,Y 312.607,Z 392.155,A -85,B 0,C 180,E1 -15675.651,E2 -15675.651} C_VEL
LIN {X 0,Y 312.524,Z 392.175,A -85,B 0,C 180,E1 -15679.714,E2 -15679.714} C_VEL
LIN {X 0,Y 312.503,Z 392.179,A -85,B 0,C 180,E1 -15682.777,E2 -15682.777} C_VEL
LIN {X 0,Y 312.469,Z 392.182,A -85,B 0,C 180,E1 -15686.733,E2 -15686.733} C_VEL
LIN {X 0,Y 312.453,Z 392.179,A -85,B 0,C 180,E1 -15689.66,E2 -15689.66} C_VEL
LIN {X 0,Y 312.507,Z 392.18,A -85,B 0,C 180,E1 -15693.69,E2 -15693.69} C_VEL
LIN {X 0,Y 312.498,Z 392.143,A -85,B 0,C 180,E1 -15697.389,E2 -15697.389} C_VEL
LIN {X 0,Y 312.475,Z 392.401,A -85,B 0,C 180,E1 -15698.699,E2 -15698.699} C_VEL
LIN {X 0,Y 313.375,Z 394.891,A -85,B 0,C 180,E1 -15699.398,E2 -15699.398} C_VEL
LIN {X 0,Y 317.261,Z 403.31,A -85,B 0,C 180,E1 -15701.649,E2 -15701.649} C_VEL
LIN {X 0,Y 322.961,Z 417.57,A -85,B 0,C 180,E1 -15705.063,E2 -15705.063} C_VEL
LIN {X 0,Y 327.679,Z 431.57,A -85,B 0,C 180,E1 -15708.083,E2 -15708.083} C_VEL
LIN {X 0,Y 331.873,Z 446.149,A -85,B 0,C 180,E1 -15710.949,E2 -15710.949} C_VEL
LIN {X 0,Y 333.273,Z 452.141,A -85,B 0,C 180,E1 -15712.047,E2 -15712.047} C_VEL
LIN {X 0,Y 331.391,Z 471.075,A -85,B 0,C 180,E1 -15714.524,E2 -15714.524} C_VEL
LIN {X 0,Y 336.525,Z 504.889,A -85,B 0,C 180,E1 -15716.014,E2 -15716.014} C_VEL
LIN {X 0,Y 337.716,Z 515.181,A -85,B 0,C 180,E1 -15716.408,E2 -15716.408} C_VEL
LIN {X 0,Y 333.415,Z 640.105,A -85,B 0,C 180,E1 -15719.086,E2 -15719.086} C_VEL
LIN {X 0,Y 332.433,Z 654.904,A -85,B 0,C 180,E1 -15719.601,E2 -15719.601} C_VEL
LIN {X 0,Y 330.909,Z 669.51,A -85,B 0,C 180,E1 -15720.325,E2 -15720.325} C_VEL
LIN {X 0,Y 329.034,Z 684.337,A -85,B 0,C 180,E1 -15721.328,E2 -15721.328} C_VEL
LIN {X 0,Y 327.057,Z 697.653,A -85,B 0,C 180,E1 -15722.486,E2 -15722.486} C_VEL
LIN {X 0,Y 324.53,Z 711.627,A -85,B 0,C 180,E1 -15723.992,E2 -15723.992} C_VEL
LIN {X 0,Y 322.109,Z 724.222,A -85,B 0,C 180,E1 -15725.683,E2 -15725.683} C_VEL
LIN {X 0,Y 319.964,Z 735.087,A -85,B 0,C 180,E1 -15727.457,E2 -15727.457} C_VEL
LIN {X 0,Y 317.516,Z 746.018,A -85,B 0,C 180,E1 -15729.6,E2 -15729.6} C_VEL
LIN {X 0,Y 315.54,Z 755.328,A -85,B 0,C 180,E1 -15731.833,E2 -15731.833} C_VEL
LIN {X 0,Y 314.113,Z 762.076,A -85,B 0,C 180,E1 -15733.761,E2 -15733.761} C_VEL
LIN {X 0,Y 312.749,Z 769.499,A -85,B 0,C 180,E1 -15736.354,E2 -15736.354} C_VEL
LIN {X 0,Y 311.678,Z 775.394,A -85,B 0,C 180,E1 -15738.952,E2 -15738.952} C_VEL
LIN {X 0,Y 311.211,Z 778.872,A -85,B 0,C 180,E1 -15740.907,E2 -15740.907} C_VEL
LIN {X 0,Y 310.809,Z 782.415,A -85,B 0,C 180,E1 -15743.51,E2 -15743.51} C_VEL
LIN {X 0,Y 310.671,Z 784.756,A -85,B 0,C 180,E1 -15746.111,E2 -15746.111} C_VEL
LIN {X 0,Y 310.604,Z 785.947,A -85,B 0,C 180,E1 -15748.705,E2 -15748.705} C_VEL
LIN {X 0,Y 310.605,Z 785.961,A -85,B 0,C 180,E1 -15751.299,E2 -15751.299} C_VEL
LIN {X 0,Y 310.675,Z 784.823,A -85,B 0,C 180,E1 -15753.893,E2 -15753.893} C_VEL
LIN {X 0,Y 310.815,Z 782.533,A -85,B 0,C 180,E1 -15756.494,E2 -15756.494} C_VEL
LIN {X 0,Y 311.209,Z 779.037,A -85,B 0,C 180,E1 -15759.097,E2 -15759.097} C_VEL
LIN {X 0,Y 311.84,Z 774.256,A -85,B 0,C 180,E1 -15761.705,E2 -15761.705} C_VEL
LIN {X 0,Y 312.993,Z 768.066,A -85,B 0,C 180,E1 -15764.302,E2 -15764.302} C_VEL
LIN {X 0,Y 314.5,Z 760.28,A -85,B 0,C 180,E1 -15766.89,E2 -15766.89} C_VEL
LIN {X 0,Y 316.262,Z 751.974,A -85,B 0,C 180,E1 -15769.136,E2 -15769.136} C_VEL
LIN {X 0,Y 318.183,Z 743.544,A -85,B 0,C 180,E1 -15771.036,E2 -15771.036} C_VEL
LIN {X 0,Y 320.296,Z 733.331,A -85,B 0,C 180,E1 -15772.969,E2 -15772.969} C_VEL
LIN {X 0,Y 322.66,Z 721.714,A -85,B 0,C 180,E1 -15774.792,E2 -15774.792} C_VEL
LIN {X 0,Y 325.163,Z 708.605,A -85,B 0,C 180,E1 -15776.475,E2 -15776.475} C_VEL
LIN {X 0,Y 327.469,Z 695.522,A -85,B 0,C 180,E1 -15777.828,E2 -15777.828} C_VEL
LIN {X 0,Y 329.62,Z 680.74,A -85,B 0,C 180,E1 -15779.052,E2 -15779.052} C_VEL
LIN {X 0,Y 331.359,Z 665.998,A -85,B 0,C 180,E1 -15779.985,E2 -15779.985} C_VEL
LIN {X 0,Y 332.782,Z 650.9,A -85,B 0,C 180,E1 -15780.676,E2 -15780.676} C_VEL
LIN {X 0,Y 333.692,Z 635.053,A -85,B 0,C 180,E1 -15781.154,E2 -15781.154} C_VEL
LIN {X 0,Y 334.434,Z 615.564,A -85,B 0,C 180,E1 -15781.562,E2 -15781.562} C_VEL
LIN {X 0,Y 334.073,Z 609.765,A -85,B 0,C 180,E1 -15781.744,E2 -15781.744} C_VEL
LIN {X 0,Y 329.844,Z 591.139,A -85,B 0,C 180,E1 -15782.668,E2 -15782.668} C_VEL
LIN {X 0,Y 329.462,Z 585.341,A -85,B 0,C 180,E1 -15782.858,E2 -15782.858} C_VEL
LIN {X 0,Y 331.777,Z 514.116,A -85,B 0,C 180,E1 -15784.415,E2 -15784.415} C_VEL
LIN {X 0,Y 327.49,Z 484.114,A -85,B 0,C 180,E1 -15785.718,E2 -15785.718} C_VEL
LIN {X 0,Y 325.463,Z 470.765,A -85,B 0,C 180,E1 -15786.36,E2 -15786.36} C_VEL
LIN {X 0,Y 326.88,Z 456.989,A -85,B 0,C 180,E1 -15788.182,E2 -15788.182} C_VEL
LIN {X 0,Y 327.087,Z 454.433,A -85,B 0,C 180,E1 -15788.546,E2 -15788.546} C_VEL
LIN {X 0,Y 323.109,Z 439.352,A -85,B 0,C 180,E1 -15791.468,E2 -15791.468} C_VEL
LIN {X 0,Y 318.948,Z 426.307,A -85,B 0,C 180,E1 -15794.264,E2 -15794.264} C_VEL
LIN {X 0,Y 313.978,Z 412.982,A -85,B 0,C 180,E1 -15797.382,E2 -15797.382} C_VEL
LIN {X 0,Y 308.92,Z 401.201,A -85,B 0,C 180,E1 -15800.431,E2 -15800.431} C_VEL
LIN {X 0,Y 305.54,Z 393.432,A -85,B 0,C 180,E1 -15802.65,E2 -15802.65} C_VEL
LIN {X 0,Y 305.466,Z 393.033,A -85,B 0,C 180,E1 -15803.638,E2 -15803.638} C_VEL
LIN {X 0,Y 305.469,Z 393.027,A -85,B 0,C 180,E1 -15806.484,E2 -15806.484} C_VEL
LIN {X 0,Y 305.553,Z 393.269,A -85,B 0,C 180,E1 -15809.971,E2 -15809.971} C_VEL
LIN {X 0,Y 306.023,Z 395.414,A -85,B 0,C 180,E1 -15810.486,E2 -15810.486} C_VEL
LIN {X 0,Y 318.995,Z 429.338,A -85,B 0,C 180,E1 -15812.593,E2 -15812.593} C_VEL
LIN {X 0,Y 314.451,Z 539.841,A -85,B 0,C 180,E1 -15816.147,E2 -15816.147} C_VEL
LIN {X 0,Y 313.87,Z 556.128,A -85,B 0,C 180,E1 -15816.943,E2 -15816.943} C_VEL
LIN {X 0,Y 313.016,Z 571.936,A -85,B 0,C 180,E1 -15817.996,E2 -15817.996} C_VEL
LIN {X 0,Y 312.01,Z 586.189,A -85,B 0,C 180,E1 -15819.221,E2 -15819.221} C_VEL
LIN {X 0,Y 310.928,Z 599.91,A -85,B 0,C 180,E1 -15820.696,E2 -15820.696} C_VEL
LIN {X 0,Y 309.777,Z 612.517,A -85,B 0,C 180,E1 -15822.343,E2 -15822.343} C_VEL
LIN {X 0,Y 308.836,Z 623.992,A -85,B 0,C 180,E1 -15824.152,E2 -15824.152} C_VEL
LIN {X 0,Y 307.876,Z 634.46,A -85,B 0,C 180,E1 -15826.132,E2 -15826.132} C_VEL
LIN {X 0,Y 307.186,Z 643.203,A -85,B 0,C 180,E1 -15828.117,E2 -15828.117} C_VEL
LIN {X 0,Y 306.544,Z 651.362,A -85,B 0,C 180,E1 -15830.355,E2 -15830.355} C_VEL
LIN {X 0,Y 306.164,Z 658.4,A -85,B 0,C 180,E1 -15832.747,E2 -15832.747} C_VEL
LIN {X 0,Y 305.7,Z 664.509,A -85,B 0,C 180,E1 -15835.385,E2 -15835.385} C_VEL
LIN {X 0,Y 305.76,Z 668.004,A -85,B 0,C 180,E1 -15837.365,E2 -15837.365} C_VEL
LIN {X 0,Y 305.875,Z 669.857,A -85,B 0,C 180,E1 -15838.683,E2 -15838.683} C_VEL
LIN {X 0,Y 305.881,Z 671.367,A -85,B 0,C 180,E1 -15840,E2 -15840} C_VEL
LIN {X 0,Y 306.274,Z 672.474,A -85,B 0,C 180,E1 -15841.315,E2 -15841.315} C_VEL
LIN {X 0,Y 306.975,Z 673.662,A -85,B 0,C 180,E1 -15843.938,E2 -15843.938} C_VEL
LIN {X 0,Y 307.851,Z 673.468,A -85,B 0,C 180,E1 -15846.554,E2 -15846.554} C_VEL
LIN {X 0,Y 309.234,Z 671.808,A -85,B 0,C 180,E1 -15849.154,E2 -15849.154} C_VEL
LIN {X 0,Y 310.928,Z 668.729,A -85,B 0,C 180,E1 -15851.737,E2 -15851.737} C_VEL
LIN {X 0,Y 313.161,Z 664.051,A -85,B 0,C 180,E1 -15854.292,E2 -15854.292} C_VEL
LIN {X 0,Y 315.822,Z 657.615,A -85,B 0,C 180,E1 -15856.883,E2 -15856.883} C_VEL
LIN {X 0,Y 318.362,Z 650.77,A -85,B 0,C 180,E1 -15859.003,E2 -15859.003} C_VEL
LIN {X 0,Y 321.283,Z 642.134,A -85,B 0,C 180,E1 -15861.157,E2 -15861.157} C_VEL
LIN {X 0,Y 324.099,Z 633.125,A -85,B 0,C 180,E1 -15862.975,E2 -15862.975} C_VEL
LIN {X 0,Y 327.51,Z 620.887,A -85,B 0,C 180,E1 -15865.007,E2 -15865.007} C_VEL
LIN {X 0,Y 330.333,Z 609.502,A -85,B 0,C 180,E1 -15866.537,E2 -15866.537} C_VEL
LIN {X 0,Y 332.919,Z 597.787,A -85,B 0,C 180,E1 -15867.844,E2 -15867.844} C_VEL
LIN {X 0,Y 335.658,Z 583.556,A -85,B 0,C 180,E1 -15869.131,E2 -15869.131} C_VEL
LIN {X 0,Y 337.858,Z 569.91,A -85,B 0,C 180,E1 -15870.122,E2 -15870.122} C_VEL
LIN {X 0,Y 339.979,Z 552.976,A -85,B 0,C 180,E1 -15871.074,E2 -15871.074} C_VEL
LIN {X 0,Y 345.598,Z 514.614,A -85,B 0,C 180,E1 -15872.738,E2 -15872.738} C_VEL
LIN {X 0,Y 353.71,Z 467.197,A -85,B 0,C 180,E1 -15874.647,E2 -15874.647} C_VEL
LIN {X 0,Y 351.804,Z 464.185,A -85,B 0,C 180,E1 -15875.804,E2 -15875.804} C_VEL
LIN {X 0,Y 350.191,Z 461.902,A -85,B 0,C 180,E1 -15876.945,E2 -15876.945} C_VEL
LIN {X 0,Y 348.6,Z 459.844,A -85,B 0,C 180,E1 -15878.335,E2 -15878.335} C_VEL
LIN {X 0,Y 346.949,Z 458.395,A -85,B 0,C 180,E1 -15880.407,E2 -15880.407} C_VEL
LIN {X 0,Y 346.131,Z 458.803,A -85,B 0,C 180,E1 -15882.671,E2 -15882.671} C_VEL
LIN {X 0,Y 346.357,Z 460.733,A -85,B 0,C 180,E1 -15884.748,E2 -15884.748} C_VEL
LIN {X 0,Y 347.354,Z 464.143,A -85,B 0,C 180,E1 -15886.686,E2 -15886.686} C_VEL
LIN {X 0,Y 348.549,Z 467.805,A -85,B 0,C 180,E1 -15888.115,E2 -15888.115} C_VEL
LIN {X 0,Y 349.923,Z 472.867,A -85,B 0,C 180,E1 -15889.487,E2 -15889.487} C_VEL
LIN {X 0,Y 349.387,Z 488.495,A -85,B 0,C 180,E1 -15890.957,E2 -15890.957} C_VEL
LIN {X 0,Y 348.706,Z 503.12,A -85,B 0,C 180,E1 -15892.077,E2 -15892.077} C_VEL
LIN {X 0,Y 347.675,Z 516.215,A -85,B 0,C 180,E1 -15892.85,E2 -15892.85} C_VEL
LIN {X 0,Y 338.594,Z 583.68,A -85,B 0,C 180,E1 -15895.328,E2 -15895.328} C_VEL
LIN {X 0,Y 335.415,Z 607.416,A -85,B 0,C 180,E1 -15896.225,E2 -15896.225} C_VEL
LIN {X 0,Y 332.338,Z 624.622,A -85,B 0,C 180,E1 -15897.095,E2 -15897.095} C_VEL
LIN {X 0,Y 328.458,Z 641.697,A -85,B 0,C 180,E1 -15898.202,E2 -15898.202} C_VEL
LIN {X 0,Y 326.108,Z 651.204,A -85,B 0,C 180,E1 -15898.942,E2 -15898.942} C_VEL
LIN {X 0,Y 324.735,Z 665.479,A -85,B 0,C 180,E1 -15899.608,E2 -15899.608} C_VEL
LIN {X 0,Y 323.038,Z 679.763,A -85,B 0,C 180,E1 -15900.522,E2 -15900.522} C_VEL
LIN {X 0,Y 320.909,Z 694.257,A -85,B 0,C 180,E1 -15901.73,E2 -15901.73} C_VEL
LIN {X 0,Y 318.558,Z 707.464,A -85,B 0,C 180,E1 -15903.109,E2 -15903.109} C_VEL
LIN {X 0,Y 315.958,Z 720.657,A -85,B 0,C 180,E1 -15904.822,E2 -15904.822} C_VEL
LIN {X 0,Y 313.698,Z 731.287,A -85,B 0,C 180,E1 -15906.49,E2 -15906.49} C_VEL
